TestEnabled909090XYZMoveVxExpectNoErrorsCorrectPosVelAcc();

TestEnabledN22N21P4XYZMoveVxVyVzExpectNoErrorsCorrectPosVelAcc();

TestEnabledN22N21P4XYZMoveVyExpectNoErrorsCorrectPosVelAcc();

ACTION AssertNoErrors:

AssertFalse(
    Condition := tonTimeout.Q,
    Message := 'Timeout timer ended the test because it took longer than expected.'
);

AssertFalse(
    Condition := stMotionStageRx.bError,
    Message := 'Rx axis error detected when it should not have an error.'
);

AssertFalse(
    Condition := stMotionStageRy.bError,
    Message := 'Ry axis error detected when it should not have an error.'
);

AssertFalse(
    Condition := stMotionStageRz.bError,
    Message := 'Rz axis error detected when it should not have an error.'
);

AssertFalse(
    Condition := stMotionStageVx.bError,
    Message := 'Vx axis error detected when it should not have an error.'
);

AssertFalse(
    Condition := stMotionStageVy.bError,
    Message := 'Vy axis error detected when it should not have an error.'
);

AssertFalse(
    Condition := stMotionStageVz.bError,
    Message := 'Vz axis error detected when it should not have an error.'
);
END_ACTION


METHOD PRIVATE AssertPosVelAccCorrect
VAR_INPUT
    fDelta : LREAL;

    fRxPosExpected : LREAL;
    fRyPosExpected : LREAL;
    fRzPosExpected : LREAL;
    fVxPosExpected : LREAL;
    fVyPosExpected : LREAL;
    fVzPosExpected : LREAL;

    fRxVelExpected : LREAL;
    fRyVelExpected : LREAL;
    fRzVelExpected : LREAL;
    fVxVelExpected : LREAL;
    fVyVelExpected : LREAL;
    fVzVelExpected : LREAL;

    fRxAccExpected : LREAL;
    fRyAccExpected : LREAL;
    fRzAccExpected : LREAL;
    fVxAccExpected : LREAL;
    fVyAccExpected : LREAL;
    fVzAccExpected : LREAL;
END_VAR

// Position
AssertEquals_LREAL(
    Expected := fRxPosExpected,
    Actual := stMotionStageRx.Axis.NcToPlc.ActPos,
    Delta := fDelta,
    Message := 'Rx did not end at expected position.'
);

AssertEquals_LREAL(
    Expected := fRyPosExpected,
    Actual := stMotionStageRy.Axis.NcToPlc.ActPos,
    Delta := fDelta,
    Message := 'Ry did not end at expected position.'
);

AssertEquals_LREAL(
    Expected := fRzPosExpected,
    Actual := stMotionStageRz.Axis.NcToPlc.ActPos,
    Delta := fDelta,
    Message := 'Rz did not end at expected position.'
);

AssertEquals_LREAL(
    Expected := fVxPosExpected,
    Actual := stMotionStageVx.Axis.NcToPlc.ActPos,
    Delta := fDelta,
    Message := 'Vx did not end at expected position.'
);

AssertEquals_LREAL(
    Expected := fVyPosExpected,
    Actual := stMotionStageVy.Axis.NcToPlc.ActPos,
    Delta := fDelta,
    Message := 'Vy did not end at expected position.'
);

AssertEquals_LREAL(
    Expected := fVzPosExpected,
    Actual := stMotionStageVz.Axis.NcToPlc.ActPos,
    Delta := fDelta,
    Message := 'Vz did not end at expected position.'
);

// Velocity
AssertEquals_LREAL(
    Expected := fRxVelExpected,
    Actual := stMotionStageRx.fVelocity,
    Delta := fDelta,
    Message := 'Rx did not use the expected velocity.'
);

AssertEquals_LREAL(
    Expected := fRyVelExpected,
    Actual := stMotionStageRy.fVelocity,
    Delta := fDelta,
    Message := 'Ry did not use the expected velocity.'
);

AssertEquals_LREAL(
    Expected := fRzVelExpected,
    Actual := stMotionStageRz.fVelocity,
    Delta := fDelta,
    Message := 'Rz did not use the expected velocity.'
);

AssertEquals_LREAL(
    Expected := fVxVelExpected,
    Actual := stMotionStageVx.fVelocity,
    Delta := fDelta,
    Message := 'Vx did not use the expected velocity.'
);

AssertEquals_LREAL(
    Expected := fVyVelExpected,
    Actual := stMotionStageVy.fVelocity,
    Delta := fDelta,
    Message := 'Vy did not use the expected velocity.'
);

AssertEquals_LREAL(
    Expected := fVzVelExpected,
    Actual := stMotionStageVz.fVelocity,
    Delta := fDelta,
    Message := 'Vz did not use the expected velocity.'
);

// Acceleration
AssertEquals_LREAL(
    Expected := fRxAccExpected,
    Actual := stMotionStageRx.fAcceleration,
    Delta := fDelta,
    Message := 'Rx did not use the expected acceleration.'
);

AssertEquals_LREAL(
    Expected := fRyAccExpected,
    Actual := stMotionStageRy.fAcceleration,
    Delta := fDelta,
    Message := 'Ry did not use the expected acceleration.'
);

AssertEquals_LREAL(
    Expected := fRzAccExpected,
    Actual := stMotionStageRz.fAcceleration,
    Delta := fDelta,
    Message := 'Rz did not use the expected acceleration.'
);

AssertEquals_LREAL(
    Expected := fVxAccExpected,
    Actual := stMotionStageVx.fAcceleration,
    Delta := fDelta,
    Message := 'Vx did not use the expected acceleration.'
);

AssertEquals_LREAL(
    Expected := fVyAccExpected,
    Actual := stMotionStageVy.fAcceleration,
    Delta := fDelta,
    Message := 'Vy did not use the expected acceleration.'
);

AssertEquals_LREAL(
    Expected := fVzAccExpected,
    Actual := stMotionStageVz.fAcceleration,
    Delta := fDelta,
    Message := 'Vz did not use the expected acceleration.'
);
END_METHOD


METHOD PRIVATE InitMotors : BOOL

fbMotorTestSuite.SetEnables(stMotionStage := stMotionStageRx);
fbMotorTestSuite.SetEnables(stMotionStage := stMotionStageRy);
fbMotorTestSuite.SetEnables(stMotionStage := stMotionStageRz);
fbMotorTestSuite.SetEnables(stMotionStage := stMotionStageVx);
fbMotorTestSuite.SetEnables(stMotionStage := stMotionStageVy);
fbMotorTestSuite.SetEnables(stMotionStage := stMotionStageVz);

SetTar0();

fbMotionStageSetHelperRx(
    bExecute := TRUE,
    fStartPosition := 0.0,
    stMotionStage := stMotionStageRx,
    bResetDone => ,
    bSetDone =>
);

fbMotionStageSetHelperRy(
    bExecute := TRUE,
    fStartPosition := 0.0,
    stMotionStage := stMotionStageRy,
    bResetDone => ,
    bSetDone =>
);

fbMotionStageSetHelperRz(
    bExecute := TRUE,
    fStartPosition := 0.0,
    stMotionStage := stMotionStageRz,
    bResetDone => ,
    bSetDone =>
);

fbMotionStageSetHelperVx(
    bExecute := TRUE,
    fStartPosition := 0.0,
    stMotionStage := stMotionStageVx,
    bResetDone => ,
    bSetDone =>
);

fbMotionStageSetHelperVy(
    bExecute := TRUE,
    fStartPosition := 0.0,
    stMotionStage := stMotionStageVy,
    bResetDone => ,
    bSetDone =>
);

fbMotionStageSetHelperVz(
    bExecute := TRUE,
    fStartPosition := 0.0,
    stMotionStage := stMotionStageVz,
    bResetDone => ,
    bSetDone =>
);

IF fbMotionStageSetHelperRx.bSetDone AND
   fbMotionStageSetHelperRy.bSetDone AND
   fbMotionStageSetHelperRz.bSetDone AND
   fbMotionStageSetHelperVx.bSetDone AND
   fbMotionStageSetHelperVy.bSetDone AND
   fbMotionStageSetHelperVz.bSetDone THEN

    fbMotionStageSetHelperRx(
        bExecute := FALSE,
        fStartPosition := 0.0,
        stMotionStage := stMotionStageRx,
        bResetDone => ,
        bSetDone =>
    );

    fbMotionStageSetHelperRy(
        bExecute := FALSE,
        fStartPosition := 0.0,
        stMotionStage := stMotionStageRy,
        bResetDone => ,
        bSetDone =>
    );

    fbMotionStageSetHelperRz(
        bExecute := FALSE,
        fStartPosition := 0.0,
        stMotionStage := stMotionStageRz,
        bResetDone => ,
        bSetDone =>
    );

    fbMotionStageSetHelperVx(
        bExecute := FALSE,
        fStartPosition := 0.0,
        stMotionStage := stMotionStageVx,
        bResetDone => ,
        bSetDone =>
    );

    fbMotionStageSetHelperVy(
        bExecute := FALSE,
        fStartPosition := 0.0,
        stMotionStage := stMotionStageVy,
        bResetDone => ,
        bSetDone =>
    );

    fbMotionStageSetHelperVz(
        bExecute := FALSE,
        fStartPosition := 0.0,
        stMotionStage := stMotionStageVz,
        bResetDone => ,
        bSetDone =>
    );

    stMotionStageRx.nEnableMode := E_StageEnableMode.ALWAYS;
    stMotionStageRy.nEnableMode := E_StageEnableMode.ALWAYS;
    stMotionStageRz.nEnableMode := E_StageEnableMode.ALWAYS;
    stMotionStageVx.nEnableMode := E_StageEnableMode.ALWAYS;
    stMotionStageVy.nEnableMode := E_StageEnableMode.ALWAYS;
    stMotionStageVz.nEnableMode := E_StageEnableMode.ALWAYS;

    IF stMotionStageRx.bAllEnable AND
        stMotionStageRy.bAllEnable AND
        stMotionStageRz.bAllEnable AND
        stMotionStageVx.bAllEnable AND
        stMotionStageVy.bAllEnable AND
        stMotionStageVz.bAllEnable THEN

        InitMotors := TRUE;
    END_IF
END_IF
END_METHOD


METHOD PRIVATE SetTar0

stMotionStageVx.fPosition := 0.0;
stMotionStageVx.fVelocity := 0.0;
stMotionStageVx.fAcceleration := 0.0;

stMotionStageVy.fPosition := 0.0;
stMotionStageVy.fVelocity := 0.0;
stMotionStageVy.fAcceleration := 0.0;

stMotionStageVz.fPosition := 0.0;
stMotionStageVz.fVelocity := 0.0;
stMotionStageVz.fAcceleration := 0.0;

stMotionStageRx.fPosition := 0.0;
stMotionStageRx.fVelocity := 0.0;
stMotionStageRx.fAcceleration := 0.0;

stMotionStageRy.fPosition := 0.0;
stMotionStageRy.fVelocity := 0.0;
stMotionStageRy.fAcceleration := 0.0;

stMotionStageRz.fPosition := 0.0;
stMotionStageRz.fVelocity := 0.0;
stMotionStageRz.fAcceleration := 0.0;
END_METHOD


METHOD PRIVATE TestEnabled000045XYZMoveVxExpectNoErrorsCorrectPosVelAcc
VAR_INST
    bInit : BOOL;
    bComplete : BOOL;
    bBusyReached : BOOL;
    rtMoveCmdOnce : R_TRIG;
    fDelta : LREAL := 1e-9;
END_VAR

TEST('TestEnabled000045XYZMoveVxExpectNoErrorsCorrectPosVelAcc');

nTestIDAssigner := nTestIDAssigner + 1;

IF nTestID <> nTestIDAssigner OR NOT tonStart.Q THEN
    RETURN;
END_IF

tonTimeout(IN := TRUE, PT := T#3s);

IF NOT bInit THEN
    bInit := InitMotors();
END_IF

IF bInit THEN
    stMotionStageVx.fPosition := 15.0;
    stMotionStageVx.fVelocity := stMotionStageVx.fPosition * 2.0 / 3.0;
    stMotionStageVx.fAcceleration := stMotionStageVx.fVelocity * 5.0;
    rtMoveCmdOnce(CLK := TRUE);
    stMotionStageVx.bMoveCmd := rtMoveCmdOnce.Q;
END_IF

fbMotionVirtualFrame(
    stMotionStageRx := stMotionStageRx,
    stMotionStageRy := stMotionStageRy,
    stMotionStageRz := stMotionStageRz,
    stMotionStageVx := stMotionStageVx,
    stMotionStageVy := stMotionStageVy,
    stMotionStageVz := stMotionStageVz,
    bEnable := TRUE,
    fAlphaDegrees := 0.0,
    fBetaDegrees := 0.0,
    fGammaDegrees := 45.0,
    sOrder := 'XYZ',
    bBaseToNew := TRUE,
    fbVirtActPositionVec3 => ,
    fbVirtActVelocityVec3 => ,
    fbVirtActAcceleraVec3 =>
);

IF stMotionStageVx.bBusy THEN
    bBusyReached := TRUE;
END_IF

IF bBusyReached AND NOT stMotionStageVx.bBusy THEN
    bComplete := TRUE;
END_IF

IF (bComplete AND
    NOT stMotionStageVx.bBusy AND
    NOT stMotionStageVy.bBusy AND
    NOT stMotionStageVz.bBusy AND
    NOT stMotionStageRx.bBusy AND
    NOT stMotionStageRy.bBusy AND
    NOT stMotionStageRz.bBusy)
    OR tonTimeout.Q THEN

    AssertNoErrors();

    AssertPosVelAccCorrect(
        fDelta := fDelta,
        fRxPosExpected := stMotionStageVx.fPosition * SQRT(2.0) / 2.0,
        fRyPosExpected := stMotionStageVx.fPosition * SQRT(2.0) / 2.0,
        fRzPosExpected := 0.0,
        fVxPosExpected := stMotionStageVx.fPosition,
        fVyPosExpected := 0.0,
        fVzPosExpected := 0.0,
        fRxVelExpected := stMotionStageVx.fVelocity * SQRT(2.0) / 2.0,
        fRyVelExpected := stMotionStageVx.fVelocity * SQRT(2.0) / 2.0,
        fRzVelExpected := 0.0,
        fVxVelExpected := stMotionStageVx.fVelocity,
        fVyVelExpected := 0.0,
        fVzVelExpected := 0.0,
        fRxAccExpected := stMotionStageVx.fAcceleration * SQRT(2.0) / 2.0,
        fRyAccExpected := stMotionStageVx.fAcceleration * SQRT(2.0) / 2.0,
        fRzAccExpected := 0.0,
        fVxAccExpected := stMotionStageVx.fAcceleration,
        fVyAccExpected := 0.0,
        fVzAccExpected := 0.0
    );

    TEST_FINISHED();

    tonTimeout(IN := FALSE);

    nTestID := nTestID + 1;
END_IF

fbMotionStageRx(stMotionStage := stMotionStageRx);
fbMotionStageRy(stMotionStage := stMotionStageRy);
fbMotionStageRz(stMotionStage := stMotionStageRz);

fbMotionStageVx(stMotionStage := stMotionStageVx);
fbMotionStageVy(stMotionStage := stMotionStageVy);
fbMotionStageVz(stMotionStage := stMotionStageVz);

nPositionCountsVx := LREAL_TO_UDINT((fbMotionVirtualFrame.fbVirtActPositionVec3.x + 100.0) * 1e6);
nPositionCountsVy := LREAL_TO_UDINT((fbMotionVirtualFrame.fbVirtActPositionVec3.y + 100.0) * 1e6);
nPositionCountsVz := LREAL_TO_UDINT((fbMotionVirtualFrame.fbVirtActPositionVec3.z + 100.0) * 1e6);
END_METHOD


METHOD PRIVATE TestEnabled000090XYZMoveVxExpectNoErrorsCorrectPosVelAcc
VAR_INST
    bInit : BOOL;
    bComplete : BOOL;
    bBusyReached : BOOL;
    rtMoveCmdOnce : R_TRIG;
    fDelta : LREAL := 1e-9;
END_VAR

TEST('TestEnabled000090XYZMoveVxExpectNoErrorsCorrectPosVelAcc');

nTestIDAssigner := nTestIDAssigner + 1;

IF nTestID <> nTestIDAssigner OR NOT tonStart.Q THEN
    RETURN;
END_IF

tonTimeout(IN := TRUE, PT := T#3s);

IF NOT bInit THEN
    bInit := InitMotors();
END_IF

IF bInit THEN
    stMotionStageVx.fPosition := 20.0;
    stMotionStageVx.fVelocity := stMotionStageVx.fPosition * 2.0 / 3.0;
    stMotionStageVx.fAcceleration := stMotionStageVx.fVelocity * 5.0;
    rtMoveCmdOnce(CLK := TRUE);
    stMotionStageVx.bMoveCmd := rtMoveCmdOnce.Q;
END_IF

fbMotionVirtualFrame(
    stMotionStageRx := stMotionStageRx,
    stMotionStageRy := stMotionStageRy,
    stMotionStageRz := stMotionStageRz,
    stMotionStageVx := stMotionStageVx,
    stMotionStageVy := stMotionStageVy,
    stMotionStageVz := stMotionStageVz,
    bEnable := TRUE,
    fAlphaDegrees := 0.0,
    fBetaDegrees := 0.0,
    fGammaDegrees := 90.0,
    sOrder := 'XYZ',
    bBaseToNew := TRUE,
    fbVirtActPositionVec3 => ,
    fbVirtActVelocityVec3 => ,
    fbVirtActAcceleraVec3 =>
);

IF stMotionStageVx.bBusy THEN
    bBusyReached := TRUE;
END_IF

IF bBusyReached AND NOT stMotionStageVx.bBusy THEN
    bComplete := TRUE;
END_IF

IF (bComplete AND
    NOT stMotionStageVx.bBusy AND
    NOT stMotionStageVy.bBusy AND
    NOT stMotionStageVz.bBusy AND
    NOT stMotionStageRx.bBusy AND
    NOT stMotionStageRy.bBusy AND
    NOT stMotionStageRz.bBusy)
    OR tonTimeout.Q THEN

    AssertNoErrors();

    AssertPosVelAccCorrect(
        fDelta := fDelta,
        fRxPosExpected := 0.0,
        fRyPosExpected := stMotionStageVx.fPosition,
        fRzPosExpected := 0.0,
        fVxPosExpected := stMotionStageVx.fPosition,
        fVyPosExpected := 0.0,
        fVzPosExpected := 0.0,
        fRxVelExpected := 0.0,
        fRyVelExpected := stMotionStageVx.fVelocity,
        fRzVelExpected := 0.0,
        fVxVelExpected := stMotionStageVx.fVelocity,
        fVyVelExpected := 0.0,
        fVzVelExpected := 0.0,
        fRxAccExpected := 0.0,
        fRyAccExpected := stMotionStageVx.fAcceleration,
        fRzAccExpected := 0.0,
        fVxAccExpected := stMotionStageVx.fAcceleration,
        fVyAccExpected := 0.0,
        fVzAccExpected := 0.0
    );

    TEST_FINISHED();

    tonTimeout(IN := FALSE);

    nTestID := nTestID + 1;
END_IF

fbMotionStageRx(stMotionStage := stMotionStageRx);
fbMotionStageRy(stMotionStage := stMotionStageRy);
fbMotionStageRz(stMotionStage := stMotionStageRz);

fbMotionStageVx(stMotionStage := stMotionStageVx);
fbMotionStageVy(stMotionStage := stMotionStageVy);
fbMotionStageVz(stMotionStage := stMotionStageVz);

nPositionCountsVx := LREAL_TO_UDINT((fbMotionVirtualFrame.fbVirtActPositionVec3.x + 100.0) * 1e6);
nPositionCountsVy := LREAL_TO_UDINT((fbMotionVirtualFrame.fbVirtActPositionVec3.y + 100.0) * 1e6);
nPositionCountsVz := LREAL_TO_UDINT((fbMotionVirtualFrame.fbVirtActPositionVec3.z + 100.0) * 1e6);
END_METHOD


METHOD PRIVATE TestEnabled009090XYZMoveVxExpectNoErrorsCorrectPosVelAcc
VAR_INST
    bInit : BOOL;
    bComplete : BOOL;
    bBusyReached : BOOL;
    rtMoveCmdOnce : R_TRIG;
    fDelta : LREAL := 1e-9;
END_VAR

TEST('TestEnabled009090XYZMoveVxExpectNoErrorsCorrectPosVelAcc');

nTestIDAssigner := nTestIDAssigner + 1;

IF nTestID <> nTestIDAssigner OR NOT tonStart.Q THEN
    RETURN;
END_IF

tonTimeout(IN := TRUE, PT := T#3s);

IF NOT bInit THEN
    bInit := InitMotors();
END_IF

IF bInit THEN
    stMotionStageVx.fPosition := 25.0;
    stMotionStageVx.fVelocity := stMotionStageVx.fPosition * 2.0 / 3.0;
    stMotionStageVx.fAcceleration := stMotionStageVx.fVelocity * 5.0;
    rtMoveCmdOnce(CLK := TRUE);
    stMotionStageVx.bMoveCmd := rtMoveCmdOnce.Q;
END_IF

fbMotionVirtualFrame(
    stMotionStageRx := stMotionStageRx,
    stMotionStageRy := stMotionStageRy,
    stMotionStageRz := stMotionStageRz,
    stMotionStageVx := stMotionStageVx,
    stMotionStageVy := stMotionStageVy,
    stMotionStageVz := stMotionStageVz,
    bEnable := TRUE,
    fAlphaDegrees := 0.0,
    fBetaDegrees := 90.0,
    fGammaDegrees := 90.0,
    sOrder := 'XYZ',
    bBaseToNew := TRUE,
    fbVirtActPositionVec3 => ,
    fbVirtActVelocityVec3 => ,
    fbVirtActAcceleraVec3 =>
);

IF stMotionStageVx.bBusy THEN
    bBusyReached := TRUE;
END_IF

IF bBusyReached AND NOT stMotionStageVx.bBusy THEN
    bComplete := TRUE;
END_IF

IF (bComplete AND
    NOT stMotionStageVx.bBusy AND
    NOT stMotionStageVy.bBusy AND
    NOT stMotionStageVz.bBusy AND
    NOT stMotionStageRx.bBusy AND
    NOT stMotionStageRy.bBusy AND
    NOT stMotionStageRz.bBusy)
    OR tonTimeout.Q THEN

    AssertNoErrors();

    AssertPosVelAccCorrect(
        fDelta := fDelta,
        fRxPosExpected := 0.0,
        fRyPosExpected := stMotionStageVx.fPosition,
        fRzPosExpected := 0.0,
        fVxPosExpected := stMotionStageVx.fPosition,
        fVyPosExpected := 0.0,
        fVzPosExpected := 0.0,
        fRxVelExpected := 0.0,
        fRyVelExpected := stMotionStageVx.fVelocity,
        fRzVelExpected := 0.0,
        fVxVelExpected := stMotionStageVx.fVelocity,
        fVyVelExpected := 0.0,
        fVzVelExpected := 0.0,
        fRxAccExpected := 0.0,
        fRyAccExpected := stMotionStageVx.fAcceleration,
        fRzAccExpected := 0.0,
        fVxAccExpected := stMotionStageVx.fAcceleration,
        fVyAccExpected := 0.0,
        fVzAccExpected := 0.0
    );

    TEST_FINISHED();

    tonTimeout(IN := FALSE);

    nTestID := nTestID + 1;
END_IF

fbMotionStageRx(stMotionStage := stMotionStageRx);
fbMotionStageRy(stMotionStage := stMotionStageRy);
fbMotionStageRz(stMotionStage := stMotionStageRz);

fbMotionStageVx(stMotionStage := stMotionStageVx);
fbMotionStageVy(stMotionStage := stMotionStageVy);
fbMotionStageVz(stMotionStage := stMotionStageVz);

nPositionCountsVx := LREAL_TO_UDINT((fbMotionVirtualFrame.fbVirtActPositionVec3.x + 100.0) * 1e6);
nPositionCountsVy := LREAL_TO_UDINT((fbMotionVirtualFrame.fbVirtActPositionVec3.y + 100.0) * 1e6);
nPositionCountsVz := LREAL_TO_UDINT((fbMotionVirtualFrame.fbVirtActPositionVec3.z + 100.0) * 1e6);
END_METHOD


METHOD PRIVATE TestEnabled909090XYZMoveVxExpectNoErrorsCorrectPosVelAcc
VAR_INST
    bInit : BOOL;
    bComplete : BOOL;
    bBusyReached : BOOL;
    rtMoveCmdOnce : R_TRIG;
    fDelta : LREAL := 1e-9;
END_VAR

TEST('TestEnabled909090XYZMoveVxExpectNoErrorsCorrectPosVelAcc');

nTestIDAssigner := nTestIDAssigner + 1;

IF nTestID <> nTestIDAssigner OR NOT tonStart.Q THEN
    RETURN;
END_IF

tonTimeout(IN := TRUE, PT := T#3s);

IF NOT bInit THEN
    bInit := InitMotors();
END_IF

IF bInit THEN
    stMotionStageVx.fPosition := 35.0;
    stMotionStageVx.fVelocity := stMotionStageVx.fPosition * 2.0 / 3.0;
    stMotionStageVx.fAcceleration := stMotionStageVx.fVelocity * 5.0;
    rtMoveCmdOnce(CLK := TRUE);
    stMotionStageVx.bMoveCmd := rtMoveCmdOnce.Q;
END_IF

fbMotionVirtualFrame(
    stMotionStageRx := stMotionStageRx,
    stMotionStageRy := stMotionStageRy,
    stMotionStageRz := stMotionStageRz,
    stMotionStageVx := stMotionStageVx,
    stMotionStageVy := stMotionStageVy,
    stMotionStageVz := stMotionStageVz,
    bEnable := TRUE,
    fAlphaDegrees := 90.0,
    fBetaDegrees := 90.0,
    fGammaDegrees := 90.0,
    sOrder := 'XYZ',
    bBaseToNew := TRUE,
    fbVirtActPositionVec3 => ,
    fbVirtActVelocityVec3 => ,
    fbVirtActAcceleraVec3 =>
);

IF stMotionStageVx.bBusy THEN
    bBusyReached := TRUE;
END_IF

IF bBusyReached AND NOT stMotionStageVx.bBusy THEN
    bComplete := TRUE;
END_IF

IF (bComplete AND
    NOT stMotionStageVx.bBusy AND
    NOT stMotionStageVy.bBusy AND
    NOT stMotionStageVz.bBusy AND
    NOT stMotionStageRx.bBusy AND
    NOT stMotionStageRy.bBusy AND
    NOT stMotionStageRz.bBusy)
    OR tonTimeout.Q THEN

    AssertNoErrors();

    AssertPosVelAccCorrect(
        fDelta := fDelta,
        fRxPosExpected := 0.0,
        fRyPosExpected := 0.0,
        fRzPosExpected := stMotionStageVx.fPosition,
        fVxPosExpected := stMotionStageVx.fPosition,
        fVyPosExpected := 0.0,
        fVzPosExpected := 0.0,
        fRxVelExpected := 0.0,
        fRyVelExpected := 0.0,
        fRzVelExpected := stMotionStageVx.fVelocity,
        fVxVelExpected := stMotionStageVx.fVelocity,
        fVyVelExpected := 0.0,
        fVzVelExpected := 0.0,
        fRxAccExpected := 0.0,
        fRyAccExpected := 0.0,
        fRzAccExpected := stMotionStageVx.fAcceleration,
        fVxAccExpected := stMotionStageVx.fAcceleration,
        fVyAccExpected := 0.0,
        fVzAccExpected := 0.0
    );

    TEST_FINISHED();

    tonTimeout(IN := FALSE);

    nTestID := nTestID + 1;
END_IF

fbMotionStageRx(stMotionStage := stMotionStageRx);
fbMotionStageRy(stMotionStage := stMotionStageRy);
fbMotionStageRz(stMotionStage := stMotionStageRz);

fbMotionStageVx(stMotionStage := stMotionStageVx);
fbMotionStageVy(stMotionStage := stMotionStageVy);
fbMotionStageVz(stMotionStage := stMotionStageVz);

nPositionCountsVx := LREAL_TO_UDINT((fbMotionVirtualFrame.fbVirtActPositionVec3.x + 100.0) * 1e6);
nPositionCountsVy := LREAL_TO_UDINT((fbMotionVirtualFrame.fbVirtActPositionVec3.y + 100.0) * 1e6);
nPositionCountsVz := LREAL_TO_UDINT((fbMotionVirtualFrame.fbVirtActPositionVec3.z + 100.0) * 1e6);
END_METHOD


METHOD PRIVATE TestEnabledN22N21P4XYZMoveVxVyVzExpectNoErrorsCorrectPosVelAcc
VAR_INST
    bInit : BOOL;
    bComplete : BOOL;
    bBusyReached : BOOL;
    rtMoveCmdOnce : R_TRIG;
    fDelta : LREAL := 1e-9;
END_VAR

TEST('TestEnabledN22N21P4XYZMoveVxVyVzExpectNoErrorsCorrectPosVelAcc');

nTestIDAssigner := nTestIDAssigner + 1;

IF nTestID <> nTestIDAssigner OR NOT tonStart.Q THEN
    RETURN;
END_IF

tonTimeout(IN := TRUE, PT := T#3s);

IF NOT bInit THEN
    bInit := InitMotors();
END_IF

IF bInit THEN
    rtMoveCmdOnce(CLK := TRUE);

    stMotionStageVx.fPosition := 15.0;
    stMotionStageVx.fVelocity := stMotionStageVx.fPosition * 2.0 / 3.0;
    stMotionStageVx.fAcceleration := stMotionStageVx.fVelocity * 5.0;
    stMotionStageVx.bMoveCmd := rtMoveCmdOnce.Q;

    stMotionStageVy.fPosition := -30.0;
    stMotionStageVy.fVelocity := ABS(stMotionStageVy.fPosition * 2.0 / 3.0);
    stMotionStageVy.fAcceleration := ABS(stMotionStageVy.fVelocity * 5.0);
    stMotionStageVy.bMoveCmd := rtMoveCmdOnce.Q;

    stMotionStageVz.fPosition := 45.0;
    stMotionStageVz.fVelocity := stMotionStageVz.fPosition * 2.0 / 3.0;
    stMotionStageVz.fAcceleration := stMotionStageVz.fVelocity * 5.0;
    stMotionStageVz.bMoveCmd := rtMoveCmdOnce.Q;
END_IF

fbMotionVirtualFrame(
    stMotionStageRx := stMotionStageRx,
    stMotionStageRy := stMotionStageRy,
    stMotionStageRz := stMotionStageRz,
    stMotionStageVx := stMotionStageVx,
    stMotionStageVy := stMotionStageVy,
    stMotionStageVz := stMotionStageVz,
    bEnable := TRUE,
    fAlphaDegrees := -22.21,
    fBetaDegrees := -20.7,
    fGammaDegrees := 3.793,
    sOrder := 'XYZ',
    bBaseToNew := FALSE,
    fbVirtActPositionVec3 => ,
    fbVirtActVelocityVec3 => ,
    fbVirtActAcceleraVec3 =>
);

IF stMotionStageVx.bBusy AND stMotionStageVy.bBusy AND stMotionStageVz.bBusy THEN
    bBusyReached := TRUE;
END_IF

IF bBusyReached AND NOT stMotionStageVx.bBusy AND NOT stMotionStageVy.bBusy AND NOT stMotionStageVz.bBusy THEN
    bComplete := TRUE;
END_IF

IF (bComplete AND
    NOT stMotionStageVx.bBusy AND
    NOT stMotionStageVy.bBusy AND
    NOT stMotionStageVz.bBusy AND
    NOT stMotionStageRx.bBusy AND
    NOT stMotionStageRy.bBusy AND
    NOT stMotionStageRz.bBusy)
    OR tonTimeout.Q THEN

    AssertNoErrors();

    AssertPosVelAccCorrect(
        fDelta := fDelta,
        fRxPosExpected := 21.732640182123049,
        fRyPosExpected := -46.323371856381527,
        fRzPosExpected := 23.061603816078627,
        fVxPosExpected := stMotionStageVx.fPosition,
        fVyPosExpected := stMotionStageVy.fPosition,
        fVzPosExpected := stMotionStageVz.fPosition,
        fRxVelExpected := 14.488426788082032,
        fRyVelExpected := 30.882247904254346,
        fRzVelExpected := 15.374402544052412,
        fVxVelExpected := stMotionStageVx.fVelocity,
        fVyVelExpected := stMotionStageVy.fVelocity,
        fVzVelExpected := stMotionStageVz.fVelocity,
        fRxAccExpected := 0.724421339404102 * 1e2,
        fRyAccExpected := 1.544112395212718 * 1e2,
        fRzAccExpected := 0.768720127202621 * 1e2,
        fVxAccExpected := stMotionStageVx.fAcceleration,
        fVyAccExpected := stMotionStageVy.fAcceleration,
        fVzAccExpected := stMotionStageVz.fAcceleration
    );

    TEST_FINISHED();

    tonTimeout(IN := FALSE);

    nTestID := nTestID + 1;
END_IF

fbMotionStageRx(stMotionStage := stMotionStageRx);
fbMotionStageRy(stMotionStage := stMotionStageRy);
fbMotionStageRz(stMotionStage := stMotionStageRz);

fbMotionStageVx(stMotionStage := stMotionStageVx);
fbMotionStageVy(stMotionStage := stMotionStageVy);
fbMotionStageVz(stMotionStage := stMotionStageVz);

nPositionCountsVx := LREAL_TO_UDINT((fbMotionVirtualFrame.fbVirtActPositionVec3.x + 100.0) * 1e6);
nPositionCountsVy := LREAL_TO_UDINT((fbMotionVirtualFrame.fbVirtActPositionVec3.y + 100.0) * 1e6);
nPositionCountsVz := LREAL_TO_UDINT((fbMotionVirtualFrame.fbVirtActPositionVec3.z + 100.0) * 1e6);
END_METHOD


METHOD PRIVATE TestEnabledN22N21P4XYZMoveVyExpectNoErrorsCorrectPosVelAcc
VAR_INST
    bInit : BOOL;
    bComplete : BOOL;
    bBusyReached : BOOL;
    rtMoveCmdOnce : R_TRIG;
    fDelta : LREAL := 1e-9;
END_VAR

TEST('TestEnabledN22N21P4XYZMoveVyExpectNoErrorsCorrectPosVelAcc');

nTestIDAssigner := nTestIDAssigner + 1;

IF nTestID <> nTestIDAssigner OR NOT tonStart.Q THEN
    RETURN;
END_IF

tonTimeout(IN := TRUE, PT := T#3s);

IF NOT bInit THEN
    bInit := InitMotors();
END_IF

IF bInit THEN
    stMotionStageVy.fPosition := 30.0;
    stMotionStageVy.fVelocity := stMotionStageVy.fPosition * 2.0 / 3.0;
    stMotionStageVy.fAcceleration := stMotionStageVy.fVelocity * 5.0;
    rtMoveCmdOnce(CLK := TRUE);
    stMotionStageVy.bMoveCmd := rtMoveCmdOnce.Q;
END_IF

fbMotionVirtualFrame(
    stMotionStageRx := stMotionStageRx,
    stMotionStageRy := stMotionStageRy,
    stMotionStageRz := stMotionStageRz,
    stMotionStageVx := stMotionStageVx,
    stMotionStageVy := stMotionStageVy,
    stMotionStageVz := stMotionStageVz,
    bEnable := TRUE,
    fAlphaDegrees := -22.21,
    fBetaDegrees := -20.7,
    fGammaDegrees := 3.793,
    sOrder := 'XYZ',
    bBaseToNew := FALSE,
    fbVirtActPositionVec3 => ,
    fbVirtActVelocityVec3 => ,
    fbVirtActAcceleraVec3 =>
);

IF stMotionStageVy.bBusy THEN
    bBusyReached := TRUE;
END_IF

IF bBusyReached AND NOT stMotionStageVy.bBusy THEN
    bComplete := TRUE;
END_IF

IF (bComplete AND
    NOT stMotionStageVx.bBusy AND
    NOT stMotionStageVy.bBusy AND
    NOT stMotionStageVz.bBusy AND
    NOT stMotionStageRx.bBusy AND
    NOT stMotionStageRy.bBusy AND
    NOT stMotionStageRz.bBusy)
    OR tonTimeout.Q THEN

    AssertNoErrors();

    AssertPosVelAccCorrect(
        fDelta := fDelta,
        fRxPosExpected := 5.836964390001455,
        fRyPosExpected := 27.448135465863341,
        fRzPosExpected := 10.608001987060069,
        fVxPosExpected := 0.0,
        fVyPosExpected := stMotionStageVy.fPosition,
        fVzPosExpected := 0.0,
        fRxVelExpected := 5.836964390001455 * 2.0 / 3.0,
        fRyVelExpected := 27.448135465863341 * 2.0 / 3.0,
        fRzVelExpected := 10.608001987060069 * 2.0 / 3.0,
        fVxVelExpected := 0.0,
        fVyVelExpected := stMotionStageVy.fVelocity,
        fVzVelExpected := 0.0,
        fRxAccExpected := 5.836964390001455 * 2.0 / 3.0 * 5.0,
        fRyAccExpected := 27.448135465863341 * 2.0 / 3.0 * 5.0,
        fRzAccExpected := 10.608001987060069 * 2.0 / 3.0 * 5.0,
        fVxAccExpected := 0.0,
        fVyAccExpected := stMotionStageVy.fAcceleration,
        fVzAccExpected := 0.0
    );

    TEST_FINISHED();

    tonTimeout(IN := FALSE);

    nTestID := nTestID + 1;
END_IF

fbMotionStageRx(stMotionStage := stMotionStageRx);
fbMotionStageRy(stMotionStage := stMotionStageRy);
fbMotionStageRz(stMotionStage := stMotionStageRz);

fbMotionStageVx(stMotionStage := stMotionStageVx);
fbMotionStageVy(stMotionStage := stMotionStageVy);
fbMotionStageVz(stMotionStage := stMotionStageVz);

nPositionCountsVx := LREAL_TO_UDINT((fbMotionVirtualFrame.fbVirtActPositionVec3.x + 100.0) * 1e6);
nPositionCountsVy := LREAL_TO_UDINT((fbMotionVirtualFrame.fbVirtActPositionVec3.y + 100.0) * 1e6);
nPositionCountsVz := LREAL_TO_UDINT((fbMotionVirtualFrame.fbVirtActPositionVec3.z + 100.0) * 1e6);
END_METHOD

END_FUNCTION_BLOCK

// Tests/FB_NCErrorFFO_Test
FUNCTION_BLOCK FB_NCErrorFFO_Test EXTENDS TcUnit.FB_TestSuite
(*
    Test the following related FBs:
    - FB_NCErrorFFO
    - FB_EncErrorFFO

    These function blocks are designed to trip the beam when there
    is an NC error reported by stMotionStage.
*)
VAR
    stMotionStage: ST_MotionStage;
    fbMotionStage: FB_MotionStage;
    fbFFHWO: FB_HardwareFFOutput := (bAutoReset := TRUE);
    fbCauseNCError: FB_CauseNCError;

    fbNCErrorFFO: FB_NCErrorFFO;
    fbEncErrorFFO: FB_EncErrorFFO;

    nTestCounter: UINT;
    bOneTestDone: BOOL;
    tonTimer: TON;
END_VAR


fbMotionStage(stMotionStage:=stMotionStage);
// Limit to drive errors so I can isolate it from the enc error
fbNCErrorFFO(
    stMotionStage:=stMotionStage,
    fbFFHWO:=fbFFHWO,
    bAutoReset:=TRUE,
    nLowErrorId:=16#4500,
    nHighErrorId:=16#45FF,
);
fbEncErrorFFO(
    stMotionStage:=stMotionStage,
    fbFFHWO:=fbFFHWO,
    bAutoReset:=TRUE,
);
// Fast fault output is TRUE when there are no issues and FALSE when there is an issue
fbFFHWO.EvaluateOutput();

TestNC(0);
TestEnc(1);

IF bOneTestDone THEN
    bOneTestDone := FALSE;
    nTestCounter := nTestCounter + 1;
    tonTimer(IN:=FALSE);
    fbCauseNCError(
        Axis:=stMotionStage.Axis,
        bExecute:=FALSE,
    );
    stMotionStage.bReset := TRUE;
    fbMotionStage(stMotionStage:=stMotionStage);
END_IF
// Use this timer to time out any tests that stall
tonTimer(
    IN:=TRUE,
    PT:=T#5s,
);

METHOD TestEnc
VAR_INPUT
    nTestID: UINT;
END_VAR
VAR_INST
    nState: UINT;
END_VAR

TEST('TestEncError');
IF nTestCounter <> nTestID THEN
    RETURN;
END_IF

CASE nState OF
    0:
        // First cycle: no error, no fault
        AssertFalse(
            stMotionStage.bError,
            'Should have had no error before running this test',
        );
        AssertTrue(
            fbFFHWO.q_xFastFaultOut,
            'Should have had no fault with no error',
        );
        nState := 1;
    1:
        // Next time: cause an error
        fbCauseNCError(
            Axis:=stMotionStage.Axis,
            bExecute:=TRUE,
            nErrorCode:=16#4467, // Invalid encoder position data
        );
END_CASE

// Wait for the fault or the timeout, then check everything
IF tonTimer.Q OR (NOT fbFFHWO.q_xFastFaultOut AND stMotionStage.nErrorID = 16#4467) THEN
    AssertFalse(
        tonTimer.Q,
        'Timeout in test',
    );
    AssertTrue(
        stMotionStage.bError,
        'Did not get motor error in error test',
    );
    AssertEquals_UDINT(
        Expected:=16#4467,
        Actual:=stMotionStage.nErrorId,
        Message:='Error causer is broken',
    );
    AssertFalse(
        fbFFHWO.q_xFastFaultOut,
        Message:='Did not cause a fast fault',
    );
    AssertFalse(
        fbNCErrorFFO.bTripped,
        Message:='Drive error FB tripped with an enc error',
    );
    AssertTrue(
        fbEncErrorFFO.bTripped,
        Message:='Enc error fb did not trip with an enc error',
    );
    bOneTestDone := TRUE;
    nState := 0;
    TEST_FINISHED();
END_IF
END_METHOD

METHOD TestNC
VAR_INPUT
    nTestID: UINT;
END_VAR
VAR_INST
    nState: UINT;
END_VAR

TEST('TestNCError');
IF nTestCounter <> nTestID THEN
    RETURN;
END_IF

CASE nState OF
    0:
        // First cycle: no error, no fault
        AssertFalse(
            stMotionStage.bError,
            'Should have had no error before running this test',
        );
        AssertTrue(
            fbFFHWO.q_xFastFaultOut,
            'Should have had no fault with no error',
        );
        nState := 1;
    1:
        // Next time: cause an error
        fbCauseNCError(
            Axis:=stMotionStage.Axis,
            bExecute:=TRUE,
            nErrorCode:=16#4550, // Position lag monitoring error code
        );
END_CASE

// Wait for the fault or the timeout, then check everything
IF tonTimer.Q OR (NOT fbFFHWO.q_xFastFaultOut AND stMotionStage.nErrorId = 16#4550) THEN
    AssertFalse(
        tonTimer.Q,
        'Timeout in test',
    );
    AssertTrue(
        stMotionStage.bError,
        'Did not get motor error in error test',
    );
    AssertEquals_UDINT(
        Expected:=16#4550,
        Actual:=stMotionStage.nErrorId,
        Message:='Error causer is broken',
    );
    AssertFalse(
        fbFFHWO.q_xFastFaultOut,
        Message:='Did not cause a fast fault',
    );
    AssertTrue(
        fbNCErrorFFO.bTripped,
        Message:='NC error FB did not trip with a drive error',
    );
    AssertFalse(
        fbEncErrorFFO.bTripped,
        Message:='Enc error tripped with a drive error',
    );
    bOneTestDone := TRUE;
    TEST_FINISHED();
END_IF
END_METHOD

END_FUNCTION_BLOCK

// Tests/FB_PerMotorFFOND_Test
FUNCTION_BLOCK FB_PerMotorFFOND_Test EXTENDS TcUnit.FB_TestSuite
(*
    FFO if an illogical motor count is passed
    FFO if any motor has what looks like an encoder error
       - We'll just simulate this without doing it legit
       - The legit test is done elsewhere
    More FFOs may be added later and these will need to be tested too
*)
VAR
END_VAR


TestBlankCount();
TestTwoMotorEncError();

METHOD TestBlankCount : BOOL
VAR_INST
    fbFFO: FB_PerMotorFFOND;
    astMotionStage: ARRAY[1..MotionConstants.MAX_STATE_MOTORS] OF ST_MotionStage;
    fbFFHWO: FB_HardwareFFOutput := (bAutoReset := TRUE);
END_VAR

TEST('TestBlankCount');

fbFFHWO.EvaluateOutput();
AssertTrue(
    fbFFHWO.q_xFastFaultOut,
    'Started with a fault',
);
fbFFO(
    astMotionStage:=astMotionStage,
    fbFFHWO:=fbFFHWO,
);
fbFFHWO.EvaluateOutput();
AssertFalse(
    fbFFHWO.q_xFastFaultOut,
    'Blank count did not fault',
);
AssertTrue(
    fbFFO.bMotorCountError,
    'Blank count did not error',
);

TEST_FINISHED();
END_METHOD

METHOD TestTwoMotorEncError : BOOL
VAR_INST
    fbFFO: FB_PerMotorFFOND;
    astMotionStage: ARRAY[1..MotionConstants.MAX_STATE_MOTORS] OF ST_MotionStage;
    fbFFHWO: FB_HardwareFFOutput := (bAutoReset := TRUE);
END_VAR

TEST('TestTwoMotorEncError');

fbFFHWO.EvaluateOutput();
AssertTrue(
    fbFFHWO.q_xFastFaultOut,
    'Started with a fault',
);
astMotionStage[2].bError := TRUE;
astMotionStage[2].nErrorId := 16#4467; // Invalid encoder position data
fbFFO(
    astMotionStage:=astMotionStage,
    fbFFHWO:=fbFFHWO,
    nActiveMotorCount:=2,
);
fbFFHWO.EvaluateOutput();
AssertFalse(
    fbFFHWO.q_xFastFaultOut,
    'Encoder error did not fault',
);

TEST_FINISHED();
END_METHOD

END_FUNCTION_BLOCK

// Tests/FB_PositionStateMove_Test
FUNCTION_BLOCK FB_PositionStateMove_Test EXTENDS FB_MotorTestSuite
(*
    Test that FB_PositionStateMove can be used to move motors to named state positions
    And that the API behaves exactly as described.
*)
VAR
    stMotionStage: ST_MotionStage;
    fbMotionStage: FB_MotionStage;
    astPositionState: ARRAY[1..GeneralConstants.MAX_STATES] OF ST_PositionState;
    afbInternal: ARRAY[1..3] OF FB_PositionStateInternal;
    stDummyPos: ST_PositionState;
    stInvalid: ST_PositionState;
    stNotUpdated: ST_PositionState;
    stUnsafe: ST_PositionState;
    fbMove: FB_PositionStateMove;

    nTestCounter: UINT;
    bOneTestDone: BOOL;
    fTestStartPos: LREAL;
    tonTimer: TON;
    tonCleanup: TON;
    nIter: DINT;
    bStatesReady: BOOL;
END_VAR


astPositionState[1].sName := 'UNO';
astPositionState[1].fPosition := 10;
astPositionState[1].fDelta := 1;
astPositionState[1].fVelocity := 10;
SetGoodState(astPositionState[1]);

astPositionState[2].sName := 'DOS';
astPositionState[2].fPosition := 20;
astPositionState[2].fDelta := 1;
astPositionState[2].fVelocity := 10;
SetGoodState(astPositionState[2]);

astPositionState[3].sName := 'TRES';
astPositionState[3].fPosition := 30;
astPositionState[3].fDelta := 1;
astPositionState[3].fVelocity := 10;
SetGoodState(astPositionState[3]);

bStatesReady := TRUE;
FOR nIter := 1 TO 3 DO
    afbInternal[nIter](
        stMotionStage:=stMotionStage,
        stPositionState:=astPositionState[nIter],
    );
    bStatesReady := bStatesReady AND astPositionState[nIter].bUpdated;
END_FOR
stInvalid.bValid := FALSE;
stInvalid.bUpdated := TRUE;
stInvalid.bMoveOk := TRUE;
stNotUpdated.bValid := TRUE;
stNotUpdated.bUpdated := FALSE;
stNotUpdated.bMoveOk := TRUE;
stUnsafe.bValid := TRUE;
stUnsafe.bUpdated := TRUE;
stUnsafe.bMoveOk := FALSE;

SetEnables(stMotionStage);
fbMotionStage(stMotionStage:=stMotionStage);

IF bStatesReady AND nTestCounter = 0 THEN
    // Don't run any tests until the states are ready
    nTestCounter := 1;
    // Warm up the motion FB with a exec false runthrough
    fbMove(
        stMotionStage:=stMotionStage,
        stPositionState:=stDummyPos,
        bExecute:=FALSE,
    );
END_IF

// Test that we can move to state 1 and the outputs are correct as we go
TestMove(1, 1, FALSE);
// Test that we can move to state 2 and the outputs are correct as we go
TestMove(2, 2, FALSE);
// Test that we can interrupt a move to state 3 by dropping bExecute
TestMove(3, 3, TRUE);
// Test that we cannot move to an invalid state
TestBadStates(4);
// Test that we need a new bExecute to start a new move if a move goes from unsafe to safe
TestMoveOk(5);

// Wait a few cycles for remaining errors to propagate
tonCleanup(IN:=bOneTestDone, PT:=T#1s);
IF tonCleanup.Q THEN
    IF fbMove.bBusy THEN
        fbMove(
            stMotionStage:=stMotionStage,
            stPositionState:=stDummyPos,
            bExecute:=FALSE,
            bReset:=FALSE,
        );
    ELSIF stMotionStage.bBusy THEN
        stMotionStage.bExecute := FALSE;
    ELSIF fbMove.bError THEN
        fbMove(
            stMotionStage:=stMotionStage,
            stPositionState:=stDummyPos,
            bExecute:=FALSE,
            bReset:=TRUE,
        );
    ELSIF stMotionStage.bError THEN
       stMotionStage.bReset := TRUE;
    ELSE
        fbMove(
            stMotionStage:=stMotionStage,
            stPositionState:=stDummyPos,
            bExecute:=FALSE,
            bReset:=FALSE,
        );
        stMotionStage.bReset := FALSE;

        bOneTestDone := FALSE;
        nTestCounter := nTestCounter + 1;
        tonTimer(IN:=FALSE);
    END_IF
END_IF
// Use this timer to time out any tests that stall
tonTimer(
    IN:=bStatesReady,
    PT:=T#5s,
);

METHOD TestBadStates
VAR_INPUT
    nTestIndex: UINT;
END_VAR
TEST(CONCAT('TestInvalid', UINT_TO_STRING(nTestIndex)));
IF nTestCounter <> nTestIndex OR bOneTestDone THEN
    RETURN;
END_IF

AssertFalse(
    fbMove.bError,
    'Started with an error',
);

fbMove(
    stMotionStage:=stMotionstage,
    stPositionState:=stInvalid,
    bExecute:=TRUE,
);

AssertTrue(
    fbMove.bError,
    'Invalid should have given an error',
);

fbMove(
    stMotionStage:=stMotionstage,
    stPositionState:=stInvalid,
    bExecute:=FALSE,
    bReset:=TRUE,
);

AssertFalse(
    fbMove.bError,
    'Started with an error',
);

fbMove(
    stMotionStage:=stMotionstage,
    stPositionState:=stNotUpdated,
    bExecute:=TRUE,
    bReset:=FALSE,
);

AssertTrue(
    fbMove.bError,
    'Not updated should have given an error',
);

fbMove(
    stMotionStage:=stMotionstage,
    stPositionState:=stNotUpdated,
    bExecute:=FALSE,
    bReset:=TRUE,
);

AssertFalse(
    fbMove.bError,
    'Started with an error',
);

fbMove(
    stMotionStage:=stMotionstage,
    stPositionState:=stUnsafe,
    bExecute:=TRUE,
    bReset:=FALSE,
);

AssertTrue(
    fbMove.bError,
    'Unsafe should have given an error',
);

bOneTestDone := TRUE;
TEST_FINISHED();
END_METHOD

METHOD TestMove
VAR_INPUT
    nTestIndex: UINT;
    nStateIndex: UINT;
    bInterrupt: BOOL;
END_VAR
VAR_INST
    bLocalInit: BOOL;
    bInterruptStarted: BOOL;
    tonBusy: TON;
END_VAR
TEST(CONCAT('TestMove', UINT_TO_STRING(nTestIndex)));
IF nTestCounter <> nTestIndex OR bOneTestDone THEN
    RETURN;
END_IF

IF NOT bLocalInit THEN
    // Starting output checks
    AssertFalse(
        Condition:=fbMove.bBusy,
        Message:='Tried to start test with busy motor',
    );
    AssertFalse(
        Condition:=fbMove.bError,
        Message:='Tried to start test with errored motor',
    );
    bLocalInit := TRUE;
END_IF

// Simulate waiting a moment before stopping
tonBusy(IN:=stMotionStage.bBusy, PT:=T#100ms);
bInterruptStarted S= bInterrupt AND tonBusy.Q;

fbMove(
    stMotionStage:=stMotionstage,
    stPositionState:=astPositionState[nStateIndex],
    bExecute:=NOT bInterruptStarted,
);

IF fbMove.bDone OR tonTimer.Q OR (bInterruptStarted AND NOT fbMove.bBusy) THEN
    AssertFalse(
        tonTimer.Q,
        'Test timed out',
    );
    IF bInterrupt THEN
        AssertFalse(
            fbMove.bAtState,
            Message:='Should have been interrupted, but made it to the goal',
        );
    ELSE
        AssertTrue(
            fbMove.bAtState,
            Message:='Did not end at the state',
        );
        AssertEquals_LREAL(
            Expected:=astPositionState[nStateIndex].fPosition,
            Actual:=stMotionStage.stAxisStatus.fActPosition,
            Delta:=0.01,
            Message:='Did not reach the goal state',
        );
    END_IF
    AssertFalse(
        fbMove.bBusy,
        Message:='Was busy while done',
    );
    AssertFalse(
        fbMove.bError,
        Message:=CONCAT('Should not end in error: ', stMotionStage.sErrorMessage),
    );

    bOneTestDone := TRUE;
    bLocalInit := FALSE;
    bInterruptStarted := FALSE;
    TEST_FINISHED();
END_IF
END_METHOD

METHOD TestMoveOk
VAR_INPUT
    nTestIndex: UINT;
END_VAR
VAR_INST
    nStep: UINT;
    fStartPos: LREAL;
    stState: ST_PositionState := (
        sName:='GOAL',
        fPosition:=135,
        fDelta:=0.5,
        fVelocity:=1,
        bValid:=TRUE,
        bMoveOk:=FALSE,
        bUpdated:=TRUE
    );
    tonInternal: TON;
    bLocalExec: BOOL;
    bLocalReset: BOOL;
END_VAR
VAR CONSTANT
    END: UINT := 999;
END_VAR
TEST('TestMoveOk');
IF nTestCounter <> nTestIndex OR bOneTestDone THEN
    RETURN;
END_IF

CASE nStep OF
    // Initial setup and checks
    0:
        fStartPos := stMotionStage.stAxisStatus.fActPosition;
        AssertFalse(
            fbMove.bError,
            'Started with a fbMove error',
        );
        AssertFalse(
            stMotionStage.bError,
            'Started with a motor error',
        );
        bLocalExec := FALSE;
        bLocalReset := FALSE;
        nStep := nStep + 1;
    // Move to a state that is bad
    1:
        stState.bMoveOk := FALSE;
        bLocalExec := TRUE;
        nStep := nStep + 1;
    // The move should have failed with an error on the FB that never propagated to the motor itself- we shouldn't have attempted the move at all
    2:
        AssertTrue(
            fbMove.bError,
            'Did not have the expected move not ok error',
        );
        AssertFalse(
            stMotionStage.bError,
            'Had a motion error, but we never should have asked for a move?',
        );
        nStep := nStep + 1;
    // Make the state no longer bad, and wait a bit
    3:
        stState.bMoveOk := TRUE;
        tonInternal(IN:=TRUE, PT:=T#500ms);
        IF tonInternal.Q THEN
            tonInternal(IN:=FALSE);
            nStep := nStep + 1;
        END_IF
    // There should be no movement still
    4:
        AssertEquals_LREAL(
            Expected:=fStartPos,
            Actual:=stMotionStage.stAxisStatus.fActPosition,
            Delta:=0.1,
            Message:='Motor moved without bReset or a new bExecute!',
        );
        // Reset the error (rising edge)
        bLocalReset := TRUE;
        nStep := nStep + 1;
    // After we reset the error, wait a bit
    5:
        // Drop for rising edges later
        bLocalReset := FALSE;
        tonInternal(IN:=TRUE, PT:=T#500ms);
        IF tonInternal.Q THEN
            tonInternal(IN:=FALSE);
            nStep := nStep + 1;
        END_IF
    // There should be no error, and STILL be no movement
    6:
        AssertFalse(
            fbMove.bError,
            'The error should be reset',
        );
        AssertEquals_LREAL(
            Expected:=fStartPos,
            Actual:=stMotionStage.stAxisStatus.fActPosition,
            Delta:=0.1,
            Message:='Motor moved without a new bExecute!',
        );
        // Set bExecute to FALSE for an upcoming rising edge. It should be TRUE at this point.
        bLocalExec := FALSE;
        nStep := nStep + 1;
    // We should be able to start a move via bExecute now
    7:
        stState.fVelocity := 2000;
        stState.fAccel := 15000;
        stState.fDecel := 15000;
        bLocalExec := TRUE;
        IF fbMove.bAtState AND stMotionStage.bDone THEN
            nStep := END;
        END_IF
END_CASE

// Run fbMove exactly once every cycle no matter what
fbMove(
    stMotionStage:=stMotionStage,
    stPositionState:=stState,
    bExecute:=bLocalExec,
    bReset:=bLocalReset,
);

IF nStep = END OR tonTimer.Q THEN
    AssertFalse(
        tonTimer.Q,
        'Test timed out',
    );
    // Check that we've reached the goal
    AssertEquals_LREAL(
        Expected:=stState.fPosition,
        Actual:=stMotionStage.stAxisStatus.fActPosition,
        Delta:=0.1,
        Message:='Motor did not reach the goal.',
    );
    bOneTestDone := TRUE;
    TEST_FINISHED();
END_IF
END_METHOD

END_FUNCTION_BLOCK

// Tests/FB_PositionStateMoveND_Test
FUNCTION_BLOCK FB_PositionStateMoveND_Test EXTENDS FB_MotorTestSuite
(*
    Test that FB_PositionStateMoveND can be used to move motors to named state positions
    And that the API behaves exactly as described.
*)
VAR
    astMotionStage: ARRAY[1..MotionConstants.MAX_STATE_MOTORS] OF ST_MotionStage;
    afbMotionStage: ARRAY[1..3] OF FB_MotionStage;
    astGoalPositions: ARRAY[1..MotionConstants.MAX_STATE_MOTORS] OF ST_PositionState;
    afbInternal: ARRAY[1..3] OF FB_PositionStateInternal;
    stDummyPos: ST_PositionState;
    fbMove: FB_PositionStateMoveND;

    bInit: BOOL;
    nTestCounter: UINT;
    bOneTestDone: BOOL;
    fTestStartPos: LREAL;
    tonTimer: TON;
    nIter: DINT;
    bStatesReady: BOOL;
END_VAR


IF NOT bInit THEN
    ResetGoals();
    bInit := TRUE;
END_IF

bStatesReady := TRUE;
FOR nIter := 1 TO 3 DO
    afbInternal[nIter](
        stMotionStage:=astMotionStage[nIter],
        stPositionState:=astGoalPositions[nIter],
    );
    bStatesReady := bStatesReady AND astGoalPositions[nIter].bUpdated;
    SetEnables(astMotionStage[nIter]);
    afbMotionStage[nIter](stMotionStage:=astMotionStage[nIter]);
END_FOR

IF bStatesReady AND nTestCounter = 0 THEN
    // Don't run any tests until the states are ready
    nTestCounter := 1;
    // Warm up the motion FB with a exec false runthrough
    fbMove(
        astMotionStage := astMotionStage,
        astPositionState := astGoalPositions,
        nActiveMotorCount := 3,
        bExecute := FALSE,
    );
END_IF

// Move to somewhere
TestMove(1, 1, 5, 10, FALSE);
// Somewhere else
TestMove(2, -10, 0, 5, FALSE);
// Interrupt on the way to the last place
TestMove(3, 0, 0, 0, TRUE);

IF bOneTestDone THEN
    bOneTestDone := FALSE;
    nTestCounter := nTestCounter + 1;
    ResetGoals();
    fbMove(
        astMotionStage := astMotionStage,
        astPositionState := astGoalPositions,
        nActiveMotorCount := 3,
        bExecute := FALSE,
        bReset := TRUE,
    );
    tonTimer(IN:=FALSE);
END_IF
// Use this timer to time out any tests that stall
tonTimer(
    IN:=bStatesReady,
    PT:=T#5s,
);

METHOD ResetGoals
VAR_INPUT
END_VAR

astGoalPositions[1].sName := 'Goal1';
astGoalPositions[1].fPosition := 0;
astGoalPositions[1].fDelta := 1;
astGoalPositions[1].fVelocity := 10;
astGoalPositions[1].bUseRawCounts := FALSE;
SetGoodState(astGoalPositions[1]);

astGoalPositions[2].sName := 'Goal2';
astGoalPositions[2].fPosition := 0;
astGoalPositions[2].fDelta := 1;
astGoalPositions[2].fVelocity := 10;
astGoalPositions[2].bUseRawCounts := FALSE;
SetGoodState(astGoalPositions[2]);

astGoalPositions[3].sName := 'Goal3';
astGoalPositions[3].fPosition := 0;
astGoalPositions[3].fDelta := 1;
astGoalPositions[3].fVelocity := 10;
astGoalPositions[3].bUseRawCounts := FALSE;
SetGoodState(astGoalPositions[3]);
END_METHOD

METHOD TestMove
VAR_INPUT
    nTestIndex: UINT;
    fMotor1Pos: LREAL;
    fMotor2Pos: LREAL;
    fMotor3Pos: LREAL;
    bInterrupt: BOOL;
END_VAR
VAR_INST
    bLocalInit: BOOL;
    bInterruptStarted: BOOL;
END_VAR
TEST(CONCAT('TestMove', UINT_TO_STRING(nTestIndex)));
IF nTestCounter <> nTestIndex THEN
    RETURN;
END_IF

IF NOT bLocalInit THEN
    // Starting output checks
    AssertFalse(
        Condition:=fbMove.bBusy,
        Message:='Tried to start test with busy motor',
    );
    AssertFalse(
        Condition:=fbMove.bError,
        Message:='Tried to start test with errored motor',
    );
    bLocalInit := TRUE;
END_IF

astGoalPositions[1].fPosition := fMotor1Pos;
astGoalPositions[2].fPosition := fMotor2Pos;
astGoalPositions[3].fPosition := fMotor3Pos;

bInterruptStarted S= bInterrupt AND astMotionStage[1].bBusy AND astMotionStage[2].bBusy AND astMotionStage[3].bBusy;
fbMove(
    astMotionStage:=astMotionStage,
    astPositionState:=astGoalPositions,
    nActiveMotorCount:=3,
    bExecute:=NOT bInterruptStarted,
);
IF fbMove.bDone OR tonTimer.Q OR (bInterruptStarted AND NOT fbMove.bBusy) THEN
    IF bInterrupt THEN
        AssertFalse(
            fbMove.bAtState,
            Message:='Should have been interrupted, but made it to the goal',
        );
    ELSE
        AssertTrue(
            fbMove.bAtState,
            Message:='Did not end at the state',
        );
        FOR nIter := 1 TO 3 DO
            AssertEquals_LREAL(
                Expected:=astGoalPositions[nIter].fPosition,
                Actual:=astMotionStage[nIter].stAxisStatus.fActPosition,
                Delta:=0.01,
                Message:='Did not reach the goal state',
            );
        END_FOR

    END_IF
    AssertFalse(
        fbMove.bBusy,
        Message:='Was busy while done',
    );
    AssertFalse(
        fbMove.bError,
        Message:='Should not end in error',
    );

    bOneTestDone := TRUE;
    TEST_FINISHED();
END_IF
END_METHOD

END_FUNCTION_BLOCK

// Tests/FB_PositionStateND_Test
FUNCTION_BLOCK FB_PositionStateND_Test EXTENDS FB_MotorTestSuite
(*
    Sanity checks for the following:
    - FB_PositionState1D
    - FB_PositionState2D
    - FB_PositionState3D
    The internals have already been tested, but we need to make sure that
    they've been put together at least somewhat sensibly.
    This FB will simply use each FB to move and check the results.

    Additional tests:
    - Regression test for issue #197 (input deadlock)
*)
VAR
    stMotionStage1: ST_MotionStage;
    stMotionStage2: ST_MotionStage;
    stMotionStage3: ST_MotionStage;
    astPositionState1: ARRAY[1..GeneralConstants.MAX_STATES] OF ST_PositionState;
    astPositionState2: ARRAY[1..GeneralConstants.MAX_STATES] OF ST_PositionState;
    astPositionState3: ARRAY[1..GeneralConstants.MAX_STATES] OF ST_PositionState;
    afbInternal: ARRAY[1..3] OF ARRAY[1..3] OF FB_PositionStateInternal;
    afbMotionStage: ARRAY[1..3] OF FB_MotionStage;

    fb_Move1D: FB_PositionState1D;
    fb_Move2D: FB_PositionState2D;
    fb_Move3D: FB_PositionState3D;

    nTestCounter: UINT;
    bOneTestDone: BOOL;
    fTestStartPos: LREAL;
    tonTimer: TON;
    nIter: DINT;
    bStatesReady: BOOL;

    eSetPos: E_TestStates;
    eGetPos: E_TestStates;
END_VAR


bStatesReady := TRUE;
FOR nIter := 1 TO 3 DO;
    astPositionState1[nIter].fPosition := nIter;
    astPositionState1[nIter].fDelta := 1;
    astPositionState1[nIter].fVelocity := 100;
    astPositionState2[nIter].fPosition := 10 + nIter;
    astPositionState2[nIter].fDelta := 1;
    astPositionState2[nIter].fVelocity := 100;
    astPositionState3[nIter].fPosition := 20 + nIter;
    astPositionState3[nIter].fDelta := 1;
    astPositionState3[nIter].fVelocity := 100;
    afbInternal[nIter][1](
        stMotionStage:=stMotionStage1,
        stPositionState:=astPositionState1[nIter],
    );
    afbInternal[nIter][2](
        stMotionStage:=stMotionStage2,
        stPositionState:=astPositionState2[nIter],
    );
    afbInternal[nIter][3](
        stMotionStage:=stMotionStage3,
        stPositionState:=astPositionState3[nIter],
    );
    SetGoodState(astPositionState1[nIter]);
    SetGoodState(astPositionState2[nIter]);
    SetGoodState(astPositionState3[nIter]);
    bStatesReady := bStatesReady AND astPositionState1[nIter].bUpdated;
    bStatesReady := bStatesReady AND astPositionState2[nIter].bUpdated;
    bStatesReady := bStatesReady AND astPositionState3[nIter].bUpdated;
END_FOR
SetEnables(stMotionStage1);
SetEnables(stMotionStage2);
SetEnables(stMotionStage3);
afbMotionStage[1](stMotionStage:=stMotionStage1);
afbMotionStage[2](stMotionStage:=stMotionStage2);
afbMotionStage[3](stMotionStage:=stMotionStage3);

IF bStatesReady AND nTestCounter = 0 THEN
    // Don't run any tests until the states are ready
    nTestCounter := 1;
    // Run all the motion FBs for one cycle to warm them up
    fb_Move1D(
        stMotionStage:=stMotionStage1,
        astPositionState:=astPositionState1,
        eEnumSet:=eSetPos,
        eEnumGet:=eGetPos,
        bEnable:=TRUE,
    );
    fb_Move2D(
        stMotionStage1:=stMotionStage1,
        stMotionStage2:=stMotionStage2,
        astPositionState1:=astPositionState1,
        astPositionState2:=astPositionState2,
        eEnumSet:=eSetPos,
        eEnumGet:=eGetPos,
        bEnable:=TRUE,
    );
    fb_Move3D(
        stMotionStage1:=stMotionStage1,
        stMotionStage2:=stMotionStage2,
        stMotionStage3:=stMotionStage3,
        astPositionState1:=astPositionState1,
        astPositionState2:=astPositionState2,
        astPositionState3:=astPositionState3,
        eEnumSet:=eSetPos,
        eEnumGet:=eGetPos,
        bEnable:=TRUE,
    );
END_IF

Test1D(1, E_TestStates.OUT);
Test1D(2, E_TestStates.TARGET1);
Test1D(3, E_TestStates.TARGET2);
Test2D(4, E_TestStates.OUT);
Test2D(5, E_TestStates.TARGET1);
Test2D(6, E_TestStates.TARGET2);
Test3D(7, E_TestStates.OUT);
Test3D(8, E_TestStates.TARGET1);
Test3D(9, E_TestStates.TARGET2);
TestInputDeadlock(10);

IF bOneTestDone THEN
    bOneTestDone := FALSE;
    nTestCounter := nTestCounter + 1;
    tonTimer(IN:=FALSE);
END_IF
// Use this timer to time out any tests that stall
tonTimer(
    IN:=bStatesReady,
    PT:=T#5s,
);

METHOD Test1D
VAR_INPUT
    nTestID: UINT;
    nState: E_TestStates;
END_VAR
VAR_INST
    nLocalInit: BOOL;
END_VAR

TEST(CONCAT('Test1D_state', DINT_TO_STRING(nState)));
IF nTestCounter <> nTestID THEN
    RETURN;
END_IF

IF NOT nLocalInit THEN
    eSetPos := nState;
    nLocalInit := TRUE;
END_IF

fb_Move1D(
    stMotionStage:=stMotionStage1,
    astPositionState:=astPositionState1,
    eEnumSet:=eSetPos,
    eEnumGet:=eGetPos,
    bEnable:=TRUE,
);
IF tonTimer.Q OR fb_Move1D.stPlcToEpics.bDone THEN
    AssertTrue(
        Condition:=fb_Move1D.stPlcToEpics.bDone,
        Message:='Done should be True after move',
    );
    AssertFalse(
        Condition:=fb_Move1D.stPlcToEpics.bBusy,
        Message:='Busy should be False after move',
    );
    AssertFalse(
        Condition:=fb_Move1D.stPlcToEpics.bError,
        Message:='Error should be False after move',
    );
    AssertEquals_DINT(
        Expected:=nState,
        Actual:=eGetPos,
        Message:='Did not get to the input state',
    );
    AssertEquals_LREAL(
        Expected:=astPositionState1[nState].fPosition,
        Actual:=stMotionStage1.stAxisStatus.fActPosition,
        Delta:=0.1,
        Message:='Did not get to the input state position',
    );
    fb_Move1D.stEpicsToPlc.bReset := TRUE;
    fb_Move1D(
        stMotionStage:=stMotionStage1,
        astPositionState:=astPositionState1,
        eEnumSet:=eSetPos,
        eEnumGet:=eGetPos,
        bEnable:=TRUE,
    );
    bOneTestDone := TRUE;
    nLocalInit := FALSE;
    TEST_FINISHED();
END_IF
END_METHOD

METHOD Test2D
VAR_INPUT
    nTestID: UINT;
    nState: E_TestStates;
END_VAR
VAR_INST
    nLocalInit: BOOL;
END_VAR

TEST(CONCAT('Test2D_state', DINT_TO_STRING(nState)));
IF nTestCounter <> nTestID THEN
    RETURN;
END_IF

IF NOT nLocalInit THEN
    eSetPos := nState;
    nLocalInit := TRUE;
END_IF

fb_Move2D(
    stMotionStage1:=stMotionStage1,
    stMotionStage2:=stMotionStage2,
    astPositionState1:=astPositionState1,
    astPositionState2:=astPositionState2,
    eEnumSet:=eSetPos,
    eEnumGet:=eGetPos,
    bEnable:=TRUE,
);
IF tonTimer.Q OR fb_Move2D.stPlcToEpics.bDone THEN
    AssertTrue(
        Condition:=fb_Move2D.stPlcToEpics.bDone,
        Message:='Done should be True after move',
    );
    AssertFalse(
        Condition:=fb_Move2D.stPlcToEpics.bBusy,
        Message:='Busy should be False after move',
    );
    AssertFalse(
        Condition:=fb_Move2D.stPlcToEpics.bError,
        Message:='Error should be False after move',
    );
    AssertEquals_DINT(
        Expected:=nState,
        Actual:=eGetPos,
        Message:='Did not get to the input state',
    );
    AssertEquals_LREAL(
        Expected:=astPositionState1[nState].fPosition,
        Actual:=stMotionStage1.stAxisStatus.fActPosition,
        Delta:=0.1,
        Message:='Did not get to the input state position for stage 1',
    );
    AssertEquals_LREAL(
        Expected:=astPositionState2[nState].fPosition,
        Actual:=stMotionStage2.stAxisStatus.fActPosition,
        Delta:=0.1,
        Message:='Did not get to the input state position for stage 2',
    );
    fb_Move2D.stEpicsToPlc.bReset := TRUE;
    fb_Move2D(
        stMotionStage1:=stMotionStage1,
        stMotionStage2:=stMotionStage2,
        astPositionState1:=astPositionState1,
        astPositionState2:=astPositionState2,
        eEnumSet:=eSetPos,
        eEnumGet:=eGetPos,
        bEnable:=TRUE,
    );
    bOneTestDone := TRUE;
    nLocalInit := FALSE;
    TEST_FINISHED();
END_IF
END_METHOD

METHOD Test3D
VAR_INPUT
    nTestID: UINT;
    nState: E_TestStates;
END_VAR
VAR_INST
    nLocalInit: BOOL;
END_VAR

TEST(CONCAT('Test3D_state', DINT_TO_STRING(nState)));
IF nTestCounter <> nTestID THEN
    RETURN;
END_IF

IF NOT nLocalInit THEN
    eSetPos := nState;
    nLocalInit := TRUE;
END_IF

fb_Move3D(
    stMotionStage1:=stMotionStage1,
    stMotionStage2:=stMotionStage2,
    stMotionStage3:=stMotionStage3,
    astPositionState1:=astPositionState1,
    astPositionState2:=astPositionState2,
    astPositionState3:=astPositionState3,
    eEnumSet:=eSetPos,
    eEnumGet:=eGetPos,
    bEnable:=TRUE,
);
IF tonTimer.Q OR fb_Move3D.stPlcToEpics.bDone THEN
    AssertTrue(
        Condition:=fb_Move3D.stPlcToEpics.bDone,
        Message:='Done should be True after move',
    );
    AssertFalse(
        Condition:=fb_Move3D.stPlcToEpics.bBusy,
        Message:='Busy should be False after move',
    );
    AssertFalse(
        Condition:=fb_Move3D.stPlcToEpics.bError,
        Message:='Error should be False after move',
    );
    AssertEquals_DINT(
        Expected:=nState,
        Actual:=eGetPos,
        Message:='Did not get to the input state',
    );
    AssertEquals_LREAL(
        Expected:=astPositionState1[nState].fPosition,
        Actual:=stMotionStage1.stAxisStatus.fActPosition,
        Delta:=0.1,
        Message:='Did not get to the input state position for stage 1',
    );
    AssertEquals_LREAL(
        Expected:=astPositionState2[nState].fPosition,
        Actual:=stMotionStage2.stAxisStatus.fActPosition,
        Delta:=0.1,
        Message:='Did not get to the input state position for stage 2',
    );
    AssertEquals_LREAL(
        Expected:=astPositionState3[nState].fPosition,
        Actual:=stMotionStage3.stAxisStatus.fActPosition,
        Delta:=0.1,
        Message:='Did not get to the input state position for stage 3',
    );
    fb_Move3D.stEpicsToPlc.bReset := TRUE;
    fb_Move3D(
        stMotionStage1:=stMotionStage1,
        stMotionStage2:=stMotionStage2,
        stMotionStage3:=stMotionStage3,
        astPositionState1:=astPositionState1,
        astPositionState2:=astPositionState2,
        astPositionState3:=astPositionState3,
        eEnumSet:=eSetPos,
        eEnumGet:=eGetPos,
        bEnable:=TRUE,
    );
    bOneTestDone := TRUE;
    nLocalInit := FALSE;
    TEST_FINISHED();
END_IF
END_METHOD

METHOD TestInputDeadlock
(*
    Regression test for issue #197

    How to reproduce the issue:
    1. Get the function block into any motion error
    2. Ask for a move while in the error state

    Then, the state mover never moves again.

    To test we will follow steps 1 and 2, then reset the error, then move.

    With our fix, our second attempt at the move (after an error reset) will succeed.
    Our first attempt will fail regardless, since you cannot move a motor that is in an error state.

    Without our fix, the motor could never be moved ever again and this move will time out.
*)
VAR_INPUT
    nTestID: UINT;
END_VAR
VAR_INST
    nTestStep: UINT := 1;
    eNewGoal: E_TestStates;
END_VAR

TEST('TestInputDeadlock');
IF nTestCounter <> nTestID THEN
    RETURN;
END_IF

CASE nTestStep OF
    // Step 1: Normal move
    1:
        // Normal move: pick any other state
        IF eGetPos = E_TestStates.OUT THEN
            eNewGoal := E_TestStates.TARGET1;
        ELSE
            eNewGoal := E_TestStates.OUT;
        END_IF
        eSetPos := eNewGoal;
        nTestStep := 2;
    // Step 2: Cause a motion error. Easiest is to just set bError to TRUE during a move.
    2:
        // Cause the error if it's time
        IF stMotionStage1.bBusy THEN
            stMotionStage1.bError := TRUE;
            stMotionStage1.nErrorId := 16#4FFF;
        ELSIF stMotionStage1.bError THEN
            nTestStep := 3;
        END_IF
     // Step 3: another normal move. This should get us into the potential bugged state.
     3:
        eSetPos := eNewGoal;
        nTestStep := 4;
    // Step 4: reset the error, which will allow fixed versions of the code to resume normal operations.
    4:
        fb_Move1D.stEpicsToPlc.bReset := TRUE;
        IF NOT stMotionStage1.bError THEN
            nTestStep := 5;
        END_IF
    // Step 5: last normal move, which will succeed if we fixed the bug.
    5:
        eSetPos := eNewGoal;
        IF eGetPos = E_TestStates.Unknown THEN
            nTestStep := 6;
        END_IF
    // Step 6: wait for the move to finish
    6:
        IF eGetPos = eNewGoal THEN
            nTestStep := 7;
        END_IF
END_CASE

fb_Move1D(
    stMotionStage:=stMotionStage1,
    astPositionState:=astPositionState1,
    eEnumSet:=eSetPos,
    eEnumGet:=eGetPos,
    bEnable:=TRUE,
);

// Timeout and checks
IF tonTimer.Q OR nTestStep = 7 THEN
    AssertFalse(
        tonTimer.Q,
        'Timeout in deadlock test',
    );
    AssertEquals_UINT(
        Expected:=eNewGoal,
        Actual:=eGetPos,
        'Did not reach a goal state in deadlock test',
    );
    fb_Move1D.stEpicsToPlc.bReset := TRUE;
    fb_Move1D(
        stMotionStage:=stMotionStage1,
        astPositionState:=astPositionState1,
        eEnumSet:=eSetPos,
        eEnumGet:=eGetPos,
        bEnable:=TRUE,
    );
    bOneTestDone := TRUE;
    TEST_FINISHED();
END_IF
END_METHOD

END_FUNCTION_BLOCK

// Tests/FB_PositionStatePMPSND_Test
FUNCTION_BLOCK FB_PositionStatePMPSND_Test EXTENDS FB_MotorTestSuite
(*
    Sanity checks for the following:
    - FB_PositionStatePMPS1D
    - FB_PositionStatePMPS2D
    - FB_PositionStatePMPS3D
    The internals have already been tested, but we need to make sure that
    they've been put together at least somewhat sensibly.
    This FB will simply use each FB to move and check the results.
    In addition to reaching the goals, we need to check the beam assertions
    and the pmps limit enables.
*)
VAR
    stMotionStage1: ST_MotionStage;
    stMotionStage2: ST_MotionStage;
    stMotionStage3: ST_MotionStage;
    astPositionState1: ARRAY[1..GeneralConstants.MAX_STATES] OF ST_PositionState;
    astPositionState2: ARRAY[1..GeneralConstants.MAX_STATES] OF ST_PositionState;
    astPositionState3: ARRAY[1..GeneralConstants.MAX_STATES] OF ST_PositionState;
    afbInternal: ARRAY[1..3] OF ARRAY[1..3] OF FB_PositionStateInternal;
    afbMotionStage: ARRAY[1..3] OF FB_MotionStage;

    astBeam: ARRAY[0..3] OF ST_DbStateParams;

    fb_Move1D: FB_PositionStatePMPS1D;
    fb_Move2D: FB_PositionStatePMPS2D;
    fb_Move3D: FB_PositionStatePMPS3D;

    nTestCounter: UINT;
    bOneTestDone: BOOL;
    fTestStartPos: LREAL;
    tonTimer: TON;
    nIter: DINT;
    bStatesReady: BOOL;

    eSetPos: E_TestStates;
    eGetPos: E_TestStates;

    fbArbiter1D: FB_Arbiter(1);
    fbArbiter2D: FB_Arbiter(2);
    fbArbiter3D: FB_Arbiter(3);

    fbSubSysIO1D: FB_DummyArbIO;
    fbSubSysIO2D: FB_DummyArbIO;
    fbSubSysIO3D: FB_DummyArbIO;

    jsonHelper: FB_PMPSJsonTestHelper;
END_VAR


bStatesReady := TRUE;
FOR nIter := 1 TO 3 DO;
    astPositionState1[nIter].fPosition := nIter;
    astPositionState1[nIter].fDelta := 0.5;
    astPositionState1[nIter].fVelocity := 100;
    SetGoodState(astPositionState1[nIter]);
    astPositionState2[nIter].fPosition := 10 + nIter;
    astPositionState2[nIter].fDelta := 0.5;
    astPositionState2[nIter].fVelocity := 100;
    SetGoodState(astPositionState2[nIter]);
    astPositionState3[nIter].fPosition := 20 + nIter;
    astPositionState3[nIter].fDelta := 0.5;
    astPositionState3[nIter].fVelocity := 100;
    SetGoodState(astPositionState3[nIter]);
    afbInternal[nIter][1](
        stMotionStage:=stMotionStage1,
        stPositionState:=astPositionState1[nIter],
    );
    afbInternal[nIter][2](
        stMotionStage:=stMotionStage2,
        stPositionState:=astPositionState2[nIter],
    );
    afbInternal[nIter][3](
        stMotionStage:=stMotionStage3,
        stPositionState:=astPositionState3[nIter],
    );
    bStatesReady := bStatesReady AND astPositionState1[nIter].bUpdated;
    bStatesReady := bStatesReady AND astPositionState2[nIter].bUpdated;
    bStatesReady := bStatesReady AND astPositionState3[nIter].bUpdated;
END_FOR
SetEnablesPMPS(stMotionStage1);
SetEnablesPMPS(stMotionStage2);
SetEnablesPMPS(stMotionStage3);
IF nTestCounter <= 3 THEN
    // Startup tests, make sure the motor is enabled so we can inspect MC_Power's output
    // Otherwise we can't snoop on the PlcToNc control DWORD since this is all 0's if disabled
    // When enabled, some of the other bits go to 1 to represent directional enables
    stMotionStage1.nEnableMode := E_StageEnableMode.ALWAYS;
    stMotionStage2.nEnableMode := E_StageEnableMode.ALWAYS;
    stMotionStage3.nEnableMode := E_StageEnableMode.ALWAYS;
ELSE
    // Otherwise, make sure the most complicated mode (and the default) works
    stMotionStage1.nEnableMode := E_StageEnableMode.DURING_MOTION;
    stMotionStage2.nEnableMode := E_StageEnableMode.DURING_MOTION;
    stMotionStage3.nEnableMode := E_StageEnableMode.DURING_MOTION;
END_IF
afbMotionStage[1](stMotionStage:=stMotionStage1);
afbMotionStage[2](stMotionStage:=stMotionStage2);
afbMotionStage[3](stMotionStage:=stMotionStage3);

astBeam[E_TestStates.Unknown].stBeamParams := PMPS_GVL.cst0RateBeam;
astBeam[E_TestStates.Unknown].nRequestAssertionID := 1;
astBeam[E_TestStates.Unknown].sPmpsState := 'trans';
astBeam[E_TestStates.OUT].stBeamParams := PMPS_GVL.cstFullBeam;
astBeam[E_TestStates.OUT].nRequestAssertionID := 2;
astBeam[E_TestStates.OUT].sPmpsState := 'out';
astBeam[E_TestStates.TARGET1].stBeamParams := PMPS_GVL.cstFullBeam;
astBeam[E_TestStates.TARGET1].stBeamParams.nTran := 0.1;
astBeam[E_TestStates.TARGET1].nRequestAssertionID := 3;
astBeam[E_TestStates.TARGET1].sPmpsState := 'target1';
astBeam[E_TestStates.TARGET2].stBeamParams := PMPS_GVL.cstFullBeam;
astBeam[E_TestStates.TARGET2].stBeamParams.nTran := 0.01;
astBeam[E_TestStates.TARGET2].nRequestAssertionID := 4;
astBeam[E_TestStates.TARGET2].sPmpsState := 'target2';

// Assign beam params to states 1
astPositionState1[E_TestStates.OUT].stPMPS := astBeam[E_TestStates.OUT];
astPositionState1[E_TestStates.TARGET1].stPMPS := astBeam[E_TestStates.TARGET1];
astPositionState1[E_TestStates.TARGET2].stPMPS := astBeam[E_TestStates.TARGET2];

// Set some names for maybe help in debug
astPositionState1[E_TestStates.OUT].sName := 'OUT';
astPositionState1[E_TestStates.TARGET1].sName := 'TARGET1';
astPositionState1[E_TestStates.TARGET2].sName := 'TARGET2';
astPositionState2[E_TestStates.OUT].sName := 'OUT';
astPositionState2[E_TestStates.TARGET1].sName := 'TARGET1';
astPositionState2[E_TestStates.TARGET2].sName := 'TARGET2';
astPositionState3[E_TestStates.OUT].sName := 'OUT';
astPositionState3[E_TestStates.TARGET1].sName := 'TARGET1';
astPositionState3[E_TestStates.TARGET2].sName := 'TARGET2';

// Load a fake json doc to be consumed by our FB
jsonHelper(
    astBeamParams:=astBeam,
    bExecute:=TRUE,
    sDevName:='test',
);

IF bStatesReady AND nTestCounter = 0 THEN
    // Don't run any tests until the states are ready
    nTestCounter := 1;
END_IF

TestStartup1D(1);
TestStartup2D(2);
TestStartup3D(3);
Test1D(4, E_TestStates.OUT);
Test1D(5, E_TestStates.TARGET1);
Test1D(6, E_TestStates.TARGET2);
Test2D(7, E_TestStates.OUT);
Test2D(8, E_TestStates.TARGET1);
Test2D(9, E_TestStates.TARGET2);
Test3D(10, E_TestStates.OUT);
Test3D(11, E_TestStates.TARGET1);
Test3D(12, E_TestStates.TARGET2);
TestToggleBPTM(13);

IF bOneTestDone THEN
    bOneTestDone := FALSE;
    nTestCounter := nTestCounter + 1;
    tonTimer(IN:=FALSE);
END_IF
// Use this timer to time out any tests that stall
tonTimer(
    IN:=bStatesReady,
    PT:=T#5s,
);

METHOD AssertMotionLims: BOOL
VAR_IN_OUT
    stMotionStage: ST_MotionStage;
    astPositionState: ARRAY[1..GeneralConstants.MAX_STATES] OF ST_PositionState;
END_VAR
VAR_INPUT
    eState: E_TestStates;
    sID: STRING;
END_VAR
VAR
    nExpected: DWORD;
END_VAR

IF F_AtPositionState(stMotionStage, astPositionState[eState]) THEN
    // Both allowed
    nExpected := 2#111;
ELSIF stMotionStage.stAxisStatus.fActPosition < astPositionState[eState].fPosition THEN
    // Only + allowed
    nExpected := 2#011;
ELSE
    // Only - allowed
    nExpected := 2#101;
END_IF

IF stMotionStage.Axis.PlcToNc.ControlDWord > 0 THEN
    AssertEquals_DWORD(
        Expected:=nExpected,
        Actual:=stMotionStage.Axis.PlcToNc.ControlDWord,
        Message:=CONCAT('Wrong control dword in test ', sID),
    );
    AssertMotionLims := TRUE;
END_IF
END_METHOD

METHOD Test1D
VAR_INPUT
    nTestID: UINT;
    eState: E_TestStates;
END_VAR
VAR_INST
    fbFFHWO: FB_HardwareFFOutput;
    bInit: BOOL;
    bLimAsserted: BOOL;
END_VAR

TEST(CONCAT('Test1D_state', UINT_TO_STRING(eState)));
IF nTestCounter <> nTestID THEN
    RETURN;
END_IF

IF NOT bInit THEN
    eSetPos := eState;
END_IF

fbSubSysIO1D(
    LA:=fbArbiter1D,
    FFO:=fbFFHWO,
);

fb_Move1D(
    stMotionStage:=stMotionStage1,
    astPositionState:=astPositionState1,
    eEnumSet:=eSetPos,
    eEnumGet:=eGetPos,
    fbFFHWO:=fbFFHWO,
    fbArbiter:=fbArbiter1D,
    bEnableMotion:=TRUE,
    bEnableBeamParams:=TRUE,
    bEnablePositionLimits:=TRUE,
    bReadDBNow:=NOT bInit,
    sDeviceName:='test',
    sTransitionKey:='trans',
);

// When ready: check that directonal enables are correct
bLimAsserted S= AssertMotionLims(stMotionStage1, astPositionState1, eState, CONCAT('1D mot 1 state ', UINT_TO_STRING(eState)));


IF NOT bInit THEN
    bInit := TRUE;
END_IF

IF tonTimer.Q OR fb_Move1D.stPlcToEpics.bDone THEN
    AssertTrue(
        bLimAsserted,
        'Skipped limit assert test',
    );
    AssertTrue(
        Condition:=fb_Move1D.stPlcToEpics.bDone,
        Message:='Done should be True after move',
    );
    AssertFalse(
        Condition:=fb_Move1D.stPlcToEpics.bBusy,
        Message:='Busy should be False after move',
    );
    AssertFalse(
        Condition:=fb_Move1D.stPlcToEpics.bError,
        Message:='Error should be False after move',
    );
    AssertEquals_UINT(
        Expected:=eState,
        Actual:=eGetPos,
        Message:='Did not get to the input state',
    );
    AssertEquals_LREAL(
        Expected:=astPositionState1[eState].fPosition,
        Actual:=stMotionStage1.stAxisStatus.fActPosition,
        Delta:=0.1,
        Message:='Did not get to the input state position',
    );
    AssertTrue(
        fbArbiter1D.CheckRequestInPool(astBeam[eState].nRequestAssertionID),
        'Destination bp should have been in the arbiter',
    );
    fb_Move1D.stEpicsToPlc.bReset := TRUE;
    fb_Move1D(
        stMotionStage:=stMotionStage1,
        astPositionState:=astPositionState1,
        eEnumSet:=eSetPos,
        eEnumGet:=eGetPos,
        fbFFHWO:=fbFFHWO,
        fbArbiter:=fbArbiter1D,
        bEnableMotion:=TRUE,
        bEnableBeamParams:=TRUE,
        bEnablePositionLimits:=TRUE,
    );
    bInit := FALSE;
    bLimAsserted := FALSE;
    bOneTestDone := TRUE;
    TEST_FINISHED();
END_IF
END_METHOD

METHOD Test2D
VAR_INPUT
    nTestID: UINT;
    eState: E_TestStates;
END_VAR
VAR_INST
    fbFFHWO: FB_HardwareFFOutput;
    bInit: BOOL;
    bLimAsserted1: BOOL;
    bLimAsserted2: BOOL;
END_VAR

TEST(CONCAT('Test2D_state', UINT_TO_STRING(eState)));
IF nTestCounter <> nTestID THEN
    RETURN;
END_IF

IF NOT bInit THEN
    eSetPos := eState;
END_IF

fbSubSysIO2D(
    LA:=fbArbiter2D,
    FFO:=fbFFHWO,
);

fb_Move2D(
    stMotionStage1:=stMotionStage1,
    stMotionStage2:=stMotionStage2,
    astPositionState1:=astPositionState1,
    astPositionState2:=astPositionState2,
    eEnumSet:=eSetPos,
    eEnumGet:=eGetPos,
    fbFFHWO:=fbFFHWO,
    fbArbiter:=fbArbiter2D,
    bEnableMotion:=TRUE,
    bEnableBeamParams:=TRUE,
    bEnablePositionLimits:=TRUE,
    bReadDBNow:=NOT bInit,
    sDeviceName:='test',
    sTransitionKey:='trans',
);

// When ready: check that directonal enables are correct
bLimAsserted1 S= AssertMotionLims(stMotionStage1, astPositionState1, eState, CONCAT('2D mot 1 state ', UINT_TO_STRING(eState)));
bLimAsserted2 S= AssertMotionLims(stMotionStage2, astPositionState2, eState, CONCAT('2D mot 2 state ', UINT_TO_STRING(eState)));

IF NOT bInit THEN
    bInit := TRUE;
END_IF

IF tonTimer.Q OR fb_Move2D.stPlcToEpics.bDone THEN
    AssertTrue(
        bLimAsserted1 AND bLimAsserted2,
        'Skipped limit assert test',
    );
    AssertTrue(
        Condition:=fb_Move2D.stPlcToEpics.bDone,
        Message:='Done should be True after move',
    );
    AssertFalse(
        Condition:=fb_Move2D.stPlcToEpics.bBusy,
        Message:='Busy should be False after move',
    );
    AssertFalse(
        Condition:=fb_Move2D.stPlcToEpics.bError,
        Message:='Error should be False after move',
    );
    AssertEquals_UINT(
        Expected:=eState,
        Actual:=eGetPos,
        Message:='Did not get to the input state',
    );
    AssertEquals_LREAL(
        Expected:=astPositionState1[eState].fPosition,
        Actual:=stMotionStage1.stAxisStatus.fActPosition,
        Delta:=0.1,
        Message:='Did not get to the input state position',
    );
    AssertEquals_LREAL(
        Expected:=astPositionState2[eState].fPosition,
        Actual:=stMotionStage2.stAxisStatus.fActPosition,
        Delta:=0.1,
        Message:='Did not get to the input state position',
    );
    AssertTrue(
        fbArbiter2D.CheckRequestInPool(astBeam[eState].nRequestAssertionID),
        'Destination bp should have been in the arbiter',
    );
    fb_Move2D.stEpicsToPlc.bReset := TRUE;
    fb_Move2D(
        stMotionStage1:=stMotionStage1,
        stMotionStage2:=stMotionStage2,
        astPositionState1:=astPositionState1,
        astPositionState2:=astPositionState2,
        eEnumSet:=eSetPos,
        eEnumGet:=eGetPos,
        fbFFHWO:=fbFFHWO,
        fbArbiter:=fbArbiter2D,
        bEnableMotion:=TRUE,
        bEnableBeamParams:=TRUE,
        bEnablePositionLimits:=TRUE,
    );
    bInit := FALSE;
    bLimAsserted1 := FALSE;
    bLimAsserted2 := FALSE;
    bOneTestDone := TRUE;
    TEST_FINISHED();
END_IF
END_METHOD

METHOD Test3D
VAR_INPUT
    nTestID: UINT;
    eState: E_TestStates;
END_VAR
VAR_INST
    fbFFHWO: FB_HardwareFFOutput;
    bInit: BOOL;
    bLimAsserted1: BOOL;
    bLimAsserted2: BOOL;
    bLimAsserted3: BOOL;
END_VAR

TEST(CONCAT('Test3D_state', UINT_TO_STRING(eState)));
IF nTestCounter <> nTestID THEN
    RETURN;
END_IF

IF NOT bInit THEN
    eSetPos := eState;
END_IF

fbSubSysIO3D(
    LA:=fbArbiter3D,
    FFO:=fbFFHWO,
);

fb_Move3D(
    stMotionStage1:=stMotionStage1,
    stMotionStage2:=stMotionStage2,
    stMotionStage3:=stMotionStage3,
    eEnumSet:=eSetPos,
    eEnumGet:=eGetPos,
    astPositionState1:=astPositionState1,
    astPositionState2:=astPositionState2,
    astPositionState3:=astPositionState3,
    fbFFHWO:=fbFFHWO,
    fbArbiter:=fbArbiter3D,
    bEnableMotion:=TRUE,
    bEnableBeamParams:=TRUE,
    bEnablePositionLimits:=TRUE,
    bReadDBNow:=NOT bInit,
    sDeviceName:='test',
    sTransitionKey:='trans',
);

// When ready: check that directonal enables are correct
bLimAsserted1 S= AssertMotionLims(stMotionStage1, astPositionState1, eState, CONCAT('3D mot 1 state ', UINT_TO_STRING(eState)));
bLimAsserted2 S= AssertMotionLims(stMotionStage2, astPositionState2, eState, CONCAT('3D mot 2 state ', UINT_TO_STRING(eState)));
bLimAsserted3 S= AssertMotionLims(stMotionStage3, astPositionState3, eState, CONCAT('3D mot 3 state ', UINT_TO_STRING(eState)));

IF NOT bInit THEN
    bInit := TRUE;
END_IF

IF tonTimer.Q OR fb_Move3D.stPlcToEpics.bDone THEN
    AssertTrue(
        bLimAsserted1 AND bLimAsserted2 AND bLimAsserted3,
        'Skipped limit assert test',
    );
    AssertTrue(
        Condition:=fb_Move3D.stPlcToEpics.bDone,
        Message:='Done should be True after move',
    );
    AssertFalse(
        Condition:=fb_Move3D.stPlcToEpics.bBusy,
        Message:='Busy should be False after move',
    );
    AssertFalse(
        Condition:=fb_Move3D.stPlcToEpics.bError,
        Message:='Error should be False after move',
    );
    AssertEquals_UINT(
        Expected:=eState,
        Actual:=eGetPos,
        Message:='Did not get to the input state',
    );
    AssertEquals_LREAL(
        Expected:=astPositionState1[eState].fPosition,
        Actual:=stMotionStage1.stAxisStatus.fActPosition,
        Delta:=0.1,
        Message:='Did not get to the input state position',
    );
    AssertEquals_LREAL(
        Expected:=astPositionState2[eState].fPosition,
        Actual:=stMotionStage2.stAxisStatus.fActPosition,
        Delta:=0.1,
        Message:='Did not get to the input state position',
    );
    AssertEquals_LREAL(
        Expected:=astPositionState3[eState].fPosition,
        Actual:=stMotionStage3.stAxisStatus.fActPosition,
        Delta:=0.1,
        Message:='Did not get to the input state position',
    );
    AssertTrue(
        fbArbiter3D.CheckRequestInPool(astBeam[eState].nRequestAssertionID),
        'Destination bp should have been in the arbiter',
    );
    fb_Move3D.stEpicsToPlc.bReset := TRUE;
    fb_Move3D(
        stMotionStage1:=stMotionStage1,
        stMotionStage2:=stMotionStage2,
        stMotionStage3:=stMotionStage3,
        astPositionState1:=astPositionState1,
        astPositionState2:=astPositionState2,
        astPositionState3:=astPositionState3,
        eEnumSet:=eSetPos,
        eEnumGet:=eGetPos,
        fbFFHWO:=fbFFHWO,
        fbArbiter:=fbArbiter3D,
        bEnableMotion:=TRUE,
        bEnableBeamParams:=TRUE,
        bEnablePositionLimits:=TRUE,
    );
    bInit := FALSE;
    bLimAsserted1 := FALSE;
    bLimAsserted2 := FALSE;
    bLimAsserted3 := FALSE;
    bOneTestDone := TRUE;
    TEST_FINISHED();
END_IF
END_METHOD

METHOD TestStartup1D
(*
    - On startup, there should be no move request
    - In this case, we start in an unknown state since (0, 0, 0) is not matching any state for any motor
    - Movement should be free but the transition assertion must be active
*)
VAR_INPUT
    nTestID: UINT;
END_VAR
VAR_INST
    fbFFHWO: FB_HardwareFFOutput;
    bInit: BOOL;
END_VAR

TEST('TestStartup1D');
IF nTestCounter <> nTestID THEN
    RETURN;
END_IF

fb_Move1D(
    stMotionStage:=stMotionStage1,
    astPositionState:=astPositionState1,
    eEnumSet:=eSetPos,
    eEnumGet:=eGetPos,
    fbFFHWO:=fbFFHWO,
    fbArbiter:=fbArbiter1D,
    bEnableMotion:=TRUE,
    bEnableBeamParams:=TRUE,
    bEnablePositionLimits:=TRUE,
    bReadDBNow:=NOT bInit,
    sDeviceName:='test',
    sTransitionKey:='trans',
);

bInit := TRUE;

// We sit in this fb for some timeout number of seconds on purpose, not an error
IF tonTimer.Q THEN
    // We should neither be busy nor done (we didn't do anything)
    AssertFalse(
        Condition:=fb_Move1D.stPlcToEpics.bDone,
        Message:='Done should be False with no move',
    );
    AssertFalse(
        Condition:=fb_Move1D.stPlcToEpics.bBusy,
        Message:='Busy should be False with no move',
    );
    // We should still be at 0,0,0
    AssertEquals_LREAL(
        Expected:=0,
        Actual:=stMotionStage1.stAxisStatus.fActPosition,
        Delta:=0.0001,
        Message:='Why did we move? motor1 should have default position',
    );
    // We should be able to move both directions, which is control word 7 (2#111)
    AssertEquals_DWORD(
        Expected:=2#111,
        Actual:=stMotionStage1.Axis.PlcToNc.ControlDWord,
        Message:='Expected full +/- enables',
    );
    AssertTrue(
        fbArbiter1D.CheckRequestInPool(astBeam[E_TestStates.Unknown].nRequestAssertionID),
        'Transition assertion ID not in pool',
    );
    bOneTestDone := TRUE;
    TEST_FINISHED();
END_IF
END_METHOD

METHOD TestStartup2D
(*
    - On startup, there should be no move request
    - Starting from (0, 0, 0) all motors should only be allowed to move +
*)
VAR_INPUT
    nTestID: UINT;
END_VAR
VAR_INST
    fbFFHWO: FB_HardwareFFOutput;
    bInit: BOOL;
END_VAR

TEST('TestStartup2D');
IF nTestCounter <> nTestID THEN
    RETURN;
END_IF

fb_Move2D(
    stMotionStage1:=stMotionStage1,
    stMotionStage2:=stMotionStage2,
    astPositionState1:=astPositionState1,
    astPositionState2:=astPositionState2,
    eEnumSet:=eSetPos,
    eEnumGet:=eGetPos,
    fbFFHWO:=fbFFHWO,
    fbArbiter:=fbArbiter2D,
    bEnableMotion:=TRUE,
    bEnableBeamParams:=TRUE,
    bEnablePositionLimits:=TRUE,
    bReadDBNow:=NOT bInit,
    sDeviceName:='test',
    sTransitionKey:='trans',
);

bInit := TRUE;

// We sit in this fb for some timeout number of seconds on purpose, not an error
IF tonTimer.Q THEN
    // We should neither be busy nor done (we didn't do anything)
    AssertFalse(
        Condition:=fb_Move2D.stPlcToEpics.bDone,
        Message:='Done should be False with no move',
    );
    AssertFalse(
        Condition:=fb_Move2D.stPlcToEpics.bBusy,
        Message:='Busy should be False with no move',
    );
    // We should still be at 0,0,0
    AssertEquals_LREAL(
        Expected:=0,
        Actual:=stMotionStage1.stAxisStatus.fActPosition,
        Delta:=0.0001,
        Message:='Why did we move? motor1 should have default position',
    );
    AssertEquals_LREAL(
        Expected:=0,
        Actual:=stMotionStage2.stAxisStatus.fActPosition,
        Delta:=0.0001,
        Message:='Why did we move? motor2 should have default position',
    );
    // We should be able to move both directions, which is control word 7 (2#111)
    AssertEquals_DWORD(
        Expected:=2#111,
        Actual:=stMotionStage1.Axis.PlcToNc.ControlDWord,
        Message:='Expected full +/- enables',
    );
    AssertEquals_DWORD(
        Expected:=2#111,
        Actual:=stMotionStage2.Axis.PlcToNc.ControlDWord,
        Message:='Expected full +/- enables',
    );
    AssertTrue(
        fbArbiter2D.CheckRequestInPool(astBeam[E_TestStates.Unknown].nRequestAssertionID),
        'Transition assertion ID not in pool',
    );
    bOneTestDone := TRUE;
    TEST_FINISHED();
END_IF
END_METHOD

METHOD TestStartup3D
(*
    - On startup, there should be no move request
    - Starting from (0, 0, 0) all motors should only be allowed to move +
*)
VAR_INPUT
    nTestID: UINT;
END_VAR
VAR_INST
    fbFFHWO: FB_HardwareFFOutput;
    bInit: BOOL;
END_VAR

TEST('TestStartup3D');
IF nTestCounter <> nTestID THEN
    RETURN;
END_IF

fb_Move3D(
    stMotionStage1:=stMotionStage1,
    stMotionStage2:=stMotionStage2,
    stMotionStage3:=stMotionStage3,
    astPositionState1:=astPositionState1,
    astPositionState2:=astPositionState2,
    astPositionState3:=astPositionState3,
    eEnumSet:=eSetPos,
    eEnumGet:=eGetPos,
    fbFFHWO:=fbFFHWO,
    fbArbiter:=fbArbiter3D,
    bEnableMotion:=TRUE,
    bEnableBeamParams:=TRUE,
    bEnablePositionLimits:=TRUE,
    bReadDBNow:=NOT bInit,
    sDeviceName:='test',
    sTransitionKey:='trans',
);

bInit := TRUE;

// We sit in this fb for some timeout number of seconds on purpose, not an error
IF tonTimer.Q THEN
    // We should neither be busy nor done (we didn't do anything)
    AssertFalse(
        Condition:=fb_Move3D.stPlcToEpics.bDone,
        Message:='Done should be False with no move',
    );
    AssertFalse(
        Condition:=fb_Move3D.stPlcToEpics.bBusy,
        Message:='Busy should be False with no move',
    );
    // We should still be at 0,0,0
    AssertEquals_LREAL(
        Expected:=0,
        Actual:=stMotionStage1.stAxisStatus.fActPosition,
        Delta:=0.0001,
        Message:='Why did we move? motor1 should have default position',
    );
    AssertEquals_LREAL(
        Expected:=0,
        Actual:=stMotionStage2.stAxisStatus.fActPosition,
        Delta:=0.0001,
        Message:='Why did we move? motor2 should have default position',
    );
    AssertEquals_LREAL(
        Expected:=0,
        Actual:=stMotionStage3.stAxisStatus.fActPosition,
        Delta:=0.0001,
        Message:='Why did we move? motor3 should have default position',
    );
    // We should be able to move both directions, which is control word 7 (2#111)
    AssertEquals_DWORD(
        Expected:=2#111,
        Actual:=stMotionStage1.Axis.PlcToNc.ControlDWord,
        Message:='Expected full +/- enables',
    );
    AssertEquals_DWORD(
        Expected:=2#111,
        Actual:=stMotionStage2.Axis.PlcToNc.ControlDWord,
        Message:='Expected full +/- enables',
    );
    AssertEquals_DWORD(
        Expected:=2#111,
        Actual:=stMotionStage3.Axis.PlcToNc.ControlDWord,
        Message:='Expected full +/- enables',
    );
    AssertTrue(
        fbArbiter3D.CheckRequestInPool(astBeam[E_TestStates.Unknown].nRequestAssertionID),
        'Transition assertion ID not in pool',
    );
    bOneTestDone := TRUE;
    TEST_FINISHED();
END_IF
END_METHOD

METHOD TestToggleBPTM
VAR_INPUT
    nTestID: UINT;
END_VAR
VAR_INST
    fbFFHWO: FB_HardwareFFOutput;
    nState: UINT;
END_VAR
TEST('TestToggleBPTM');
IF nTestCounter <> nTestID THEN
    RETURN;
END_IF

fbSubSysIO1D(
    LA:=fbArbiter1D,
    FFO:=fbFFHWO,
);

IF tonTimer.Q THEN
    nState := 3;
END_IF

eSetPos := 2;

CASE nState OF
    0:
        fb_Move1D(
            stMotionStage:=stMotionStage1,
            astPositionState:=astPositionState1,
            eEnumSet:= eSetPos,
            eEnumGet:=eGetPos,
            fbFFHWO:=fbFFHWO,
            fbArbiter:=fbArbiter1D,
            bEnableMotion:=TRUE,
            bEnableBeamParams:=TRUE,
            bEnablePositionLimits:=TRUE,
            bReadDBNow:=TRUE,
            sDeviceName:='test',
            sTransitionKey:='trans',
        );
        IF fb_Move1D.stPlcToEpics.bDone THEN
            AssertTrue(
                fbArbiter1D.CheckRequestInPool(astBeam[E_TestStates.TARGET1].nRequestAssertionID),
                'Destination bp should have been in the arbiter1',
            );
            nState := 1;
        END_IF
    1:
        fb_Move1D.stPMPSEpicsToPlc.bArbiterEnabled := FALSE;
        fb_Move1D(
            stMotionStage:=stMotionStage1,
            astPositionState:=astPositionState1,
            eEnumSet:= eSetPos,
            eEnumGet:=eGetPos,
            fbFFHWO:=fbFFHWO,
            fbArbiter:=fbArbiter1D,
            bEnableMotion:=TRUE,
            bEnableBeamParams:=TRUE,
            bEnablePositionLimits:=TRUE,
            bReadDBNow:=FALSE,
            sDeviceName:='test',
            sTransitionKey:='trans',
        );
        IF fb_Move1D.stPlcToEpics.bDone THEN
            AssertFalse(
                fbArbiter1D.CheckRequestInPool(astBeam[E_TestStates.TARGET1].nRequestAssertionID),
                'Destination bp should not have been in the arbiter2',
            );
            nState := 2;
        END_IF
    2:
        fb_Move1D.stPMPSEpicsToPlc.bArbiterEnabled := TRUE;
        fb_Move1D(
            stMotionStage:=stMotionStage1,
            astPositionState:=astPositionState1,
            eEnumSet:= eSetPos,
            eEnumGet:=eGetPos,
            fbFFHWO:=fbFFHWO,
            fbArbiter:=fbArbiter1D,
            bEnableMotion:=TRUE,
            bEnableBeamParams:=TRUE,
            bEnablePositionLimits:=TRUE,
            bReadDBNow:=FALSE,
            sDeviceName:='test',
            sTransitionKey:='trans',
        );
        IF fb_Move1D.fbPMPSCore.fbMotionBPTM.bptm.eBPTMState = E_BPTMState.WaitForBP THEN
            AssertTrue(
                fbArbiter1D.CheckRequestInPool(astBeam[E_TestStates.TARGET1].nRequestAssertionID),
                'Destination bp should have been in the arbiter3',
            );
            nState := 3;
        END_IF
    3:
        AssertFalse(
            tonTimer.Q,
            'Timeout in test',
        );
        TEST_FINISHED();
END_CASE
END_METHOD

END_FUNCTION_BLOCK

// Tests/FB_PositionStateRead_Test
FUNCTION_BLOCK FB_PositionStateRead_Test EXTENDS TcUnit.FB_TestSuite
(*
    Test that FB_PositionStateRead works exactly how it should
    according to its API during normal and failure states.
*)
VAR
    stMotionStage: ST_MotionStage;
    fbMotionStage: FB_MotionStage;
    astPositionState: ARRAY[1..GeneralConstants.MAX_STATES] OF ST_PositionState;
    afbInternal: ARRAY[1..3] OF FB_PositionStateInternal;
    stDummyPos: ST_PositionState;
    fbTestMove: FB_TestHelperSetAndMove;
    fbRead: FB_PositionStateRead;

    nTestCounter: UINT;
    bOneTestDone: BOOL;
    fTestStartPos: LREAL;
    tonTimer: TON;
    nIter: DINT;
    bStatesReady: BOOL;
END_VAR


astPositionState[1].sName := 'UNO';
astPositionState[1].fPosition := 10;
astPositionState[1].fDelta := 1;
astPositionState[1].bValid := TRUE;
astPositionState[1].bUseRawCounts := FALSE;

astPositionState[2].sName := 'DOS';
astPositionState[2].fPosition := 20;
astPositionState[2].fDelta := 1;
astPositionState[2].bValid := FALSE;
astPositionState[2].bUseRawCounts := FALSE;

astPositionState[3].sName := 'TRES';
astPositionState[3].fPosition := 30;
astPositionState[3].fDelta := 1;
astPositionState[3].bValid := TRUE;
astPositionState[3].bUseRawCounts := FALSE;

astPositionState[4].sName := 'QUATRO';
astPositionState[4].fPosition := 30;
astPositionState[4].fDelta := 1;
astPositionState[4].bValid := FALSE;
astPositionState[4].bUseRawCounts := FALSE;

bStatesReady := TRUE;
FOR nIter := 1 TO 4 DO
    afbInternal[nIter](
        stMotionStage:=stMotionStage,
        stPositionState:=astPositionState[nIter],
    );
    bStatesReady := bStatesReady AND astPositionState[nIter].bUpdated;
END_FOR
fbMotionStage(stMotionStage:=stMotionStage);

// At position 1 check
TestStaticPosition(
    nTestIndex:=0,
    sTestName:='AtPos1',
    fPosition:=astPositionState[1].fPosition + 0.2 * astPositionState[1].fDelta,
    bKnownState:=TRUE,
    bMovingState:=FALSE,
    nPositionIndex:=1,
    stCurrentPosition:=astPositionState[1],
);
// Outside the deltas check
TestStaticPosition(
    nTestIndex:=1,
    sTestName:='OutsidePos1Delta',
    fPosition:=astPositionState[1].fPosition + 2 * astPositionState[1].fDelta,
    bKnownState:=FALSE,
    bMovingState:=FALSE,
    nPositionIndex:=0,
    stCurrentPosition:=stDummyPos,
);
// At invalid state 2 check
TestStaticPosition(
    nTestIndex:=2,
    sTestName:='AtInvalidPos',
    fPosition:=astPositionState[2].fPosition,
    bKnownState:=FALSE,
    bMovingState:=FALSE,
    nPositionIndex:=0,
    stCurrentPosition:=stDummyPos,
);
// At position 3 check
TestStaticPosition(
    nTestIndex:=3,
    sTestName:='AtPos3',
    fPosition:=astPositionState[3].fPosition - 0.5 * astPositionState[3].fDelta,
    bKnownState:=TRUE,
    bMovingState:=FALSE,
    nPositionIndex:=3,
    stCurrentPosition:=astPositionState[3],
);
// At position 3 and moving within bounds check
TestMovingPosition(
    nTestIndex:=4,
    sTestName:='MovingAt3',
    fStartPosition:=astPositionState[3].fPosition,
    fGoalPosition:=astPositionState[3].fPosition + 0.9 * astPositionState[3].fDelta,
    fVelocity:=0.001,
    bKnownState:=TRUE,
    bMovingState:=FALSE,
    nPositionIndex:=3,
    stCurrentPosition:=astPositionState[3],
);
// At position 3 and moving away check
TestMovingPosition(
    nTestIndex:=5,
    sTestName:='MovingFrom3',
    fStartPosition:=astPositionState[3].fPosition,
    fGoalPosition:=astPositionState[3].fPosition + 100 * astPositionState[3].fDelta,
    fVelocity:=0.001,
    bKnownState:=FALSE,
    bMovingState:=TRUE,
    nPositionIndex:=0,
    stCurrentPosition:=stDummyPos,
);
TestDupe(nTestIndex:=6);

IF bOneTestDone THEN
    bOneTestDone := FALSE;
    nTestCounter := nTestCounter + 1;
    fbTestMove(
        stMotionStage:=stMotionStage,
        bExecute:=FALSE,
    );
END_IF

METHOD PRIVATE Asserts
VAR_INPUT
    tTimeout: TIME;
    bKnownState: BOOL;
    bMovingState: BOOL;
    nPositionIndex: DINT;
    stCurrentPosition: ST_PositionState;
END_VAR
VAR
    abExpected: ARRAY[1..GeneralConstants.MAX_STATES] OF BOOL;
END_VAR

fbRead(
    stMotionStage:=stMotionStage,
    astPositionState:=astPositionstate,
);

AssertEquals_BOOL(
    Expected:=FALSE,
    Actual:=fbTestMove.tElapsed > tTimeout,
    Message:='Test timed out',
);
AssertEquals_BOOL(
    Expected:=bKnownState,
    Actual:=fbRead.bKnownState,
    Message:='Incorrect bKnownState',
);
AssertEquals_BOOL(
    Expected:=bMovingState,
    Actual:=fbRead.bMovingState,
    Message:='Incorrect bMovingState',
);
AssertEquals_DINT(
    Expected:=nPositionIndex,
    Actual:=fbRead.nPositionIndex,
    Message:='Incorrect nPositionIndex',
);
IF nPositionIndex > 0 THEN
    IF nPositionIndex <= GeneralConstants.MAX_STATES THEN
        abExpected[nPositionIndex] := TRUE;
    END_IF
 END_IF
AssertArrayEquals_BOOL(
    Expecteds:=abExpected,
    Actuals:=fbRead.abAtPosition,
    Message:='Wrong at position array',
);

IF bKnownState THEN
    AssertEquals_STRING(
        Expected:=stCurrentPosition.sName,
        Actual:=fbRead.stCurrentPosition.sName,
        Message:='Did not provide correct current position struct',
    );
END_IF
END_METHOD

METHOD TestDupe
VAR_INPUT
    nTestIndex: DINT;
END_VAR
VAR
    abExpected: ARRAY[1..GeneralConstants.MAX_STATES] OF BOOL;
END_VAR

TEST('TestDupe');
IF nTestIndex <> nTestCounter THEN
    RETURN;
END_IF

// In this test, and only in this test, we must make sure state 4 is valid
astPositionState[4].bValid := TRUE;

fbTestMove(
    stMotionStage:=stMotionStage,
    bExecute:=TRUE,
    fStartPosition:=astPositionState[4].fPosition,
    fGoalPosition:=astPositionState[4].fPosition,
);
abExpected[3] := TRUE;
abExpected[4] := TRUE;

IF fbTestMove.tElapsed > T#1s OR (fbTestMove.bSetDone AND bStatesReady) THEN
    fbRead(
        stMotionStage:=stMotionStage,
        astPositionState:=astPositionstate,
    );
    AssertEquals_BOOL(
        Expected:=FALSE,
        Actual:=fbTestMove.tElapsed > T#1s,
        Message:='Test timed out',
    );
    AssertEquals_BOOL(
        Expected:=TRUE,
        Actual:=fbRead.bKnownState,
        Message:='Incorrect bKnownState',
    );
    AssertArrayEquals_BOOL(
        Expecteds:=abExpected,
        Actuals:=fbRead.abAtPosition,
        Message:='Wrong at position array',
    );
    bOneTestDone := TRUE;
    TEST_FINISHED();
END_IF
END_METHOD

METHOD PRIVATE TestMovingPosition
VAR_INPUT
    nTestIndex: UINT;
    sTestName: STRING;
    fStartPosition: LREAL;
    fGoalPosition: LREAL;
    fVelocity: LREAL;
    bKnownState: BOOL;
    bMovingState: BOOL;
    nPositionIndex: DINT;
    stCurrentPosition: ST_PositionState;
END_VAR

TEST(sTestName);
IF nTestIndex <> nTestCounter THEN
    RETURN;
END_IF

fbTestMove(
    stMotionStage:=stMotionStage,
    bExecute:=TRUE,
    fStartPosition:=fStartPosition,
    fGoalPosition:=fGoalPosition,
    fVelocity:=0.001,
    bHWEnable:=TRUE,
);

IF fbTestMove.tElapsed > T#5s OR (fbTestMove.bMotionStarted AND bStatesReady) THEN
    Asserts(
        tTimeout:=T#5s,
        bKnownState:=bKnownState,
        bMovingState:=bMovingState,
        nPositionIndex:=nPositionIndex,
        stCurrentPosition:=stCurrentPosition,
    );
    bOneTestDone := TRUE;
    TEST_FINISHED();
END_IF
END_METHOD

METHOD PRIVATE TestStaticPosition
VAR_INPUT
    nTestIndex: UINT;
    sTestName: STRING;
    fPosition: LREAL;
    bKnownState: BOOL;
    bMovingState: BOOL;
    nPositionIndex: DINT;
    stCurrentPosition: ST_PositionState;
END_VAR

TEST(sTestName);
IF nTestIndex <> nTestCounter THEN
    RETURN;
END_IF

fbTestMove(
    stMotionStage:=stMotionStage,
    bExecute:=TRUE,
    fStartPosition:=fPosition,
    fGoalPosition:=fPosition,
);

IF fbTestMove.tElapsed > T#1s OR (fbTestMove.bSetDone AND bStatesReady) THEN
    Asserts(
        tTimeout:=T#1s,
        bKnownState:=bKnownState,
        bMovingState:=bMovingState,
        nPositionIndex:=nPositionIndex,
        stCurrentPosition:=stCurrentPosition,
    );
    bOneTestDone := TRUE;
    TEST_FINISHED();
END_IF
END_METHOD

END_FUNCTION_BLOCK

// Tests/FB_PositionStateReadND_Test
FUNCTION_BLOCK FB_PositionStateReadND_Test EXTENDS FB_MotorTestSuite
(*
    Test that FB_PositionStateReadND can be used to read and summarize
    N-dimensional state positions where multiple motors must move in
    sync to a shared named state.
*)
VAR
    astMotionStage: ARRAY[1..MotionConstants.MAX_STATE_MOTORS] OF ST_MotionStage;
    afbMotionStage: ARRAY[1..3] OF FB_MotionStage;
    astPositionState: ARRAY[1..MotionConstants.MAX_STATE_MOTORS] OF ARRAY [1..GeneralConstants.MAX_STATES] OF ST_PositionState;
    afbInternal: ARRAY[1..3] OF ARRAY [1..2] OF FB_PositionStateInternal;

    afbTestMove: ARRAY[1..3] OF FB_TestHelperSetAndMove;
    fbRead: FB_PositionStateReadND;
    bOneAssertDone: BOOL;
    nAssertCounter: UINT;
    nIter1: UINT;
    nIter2: UINT;
    nIter3: UINT;

    fbMisRead: FB_PositionStateReadND;
    astGoodStage: ARRAY[1..MotionConstants.MAX_STATE_MOTORS] OF ST_MotionStage;
    astGoodStateShape: ARRAY[1..MotionConstants.MAX_STATE_MOTORS] OF ARRAY [1..GeneralConstants.MAX_STATES] OF ST_PositionState;

    astSqMotionStage: ARRAY[1..MotionConstants.MAX_STATE_MOTORS] OF ST_MotionStage;
    afbSqMotionStage: ARRAY[1..2] OF FB_MotionStage;
    astSquareStates: ARRAY[1..MotionConstants.MAX_STATE_MOTORS] OF ARRAY [1..GeneralConstants.MAX_STATES] OF ST_PositionState;
    afbSqInternal: ARRAY[1..2] OF ARRAY[1..4] OF FB_PositionStateInternal;

